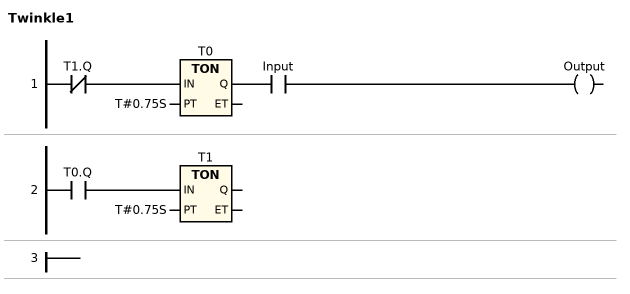
[picture p120: Twinkle1 (LD)]
_LD_ (* Ladder Diagram *)
NETWORK 1
	[/T1.Q] - T0:TON(IN: *, PT: T#0.75S) - [Input] --- (Output)
NETWORK 2
	[T0.Q] - T1:TON(IN: *, PT: T#0.75S)
NETWORK 3
	*
_END_LD_
(* the same logic as Structured Text *)
(* Network 1 *)
T0(IN := NOT T1.Q, PT := T#0.75S);
Output := T0.Q AND Input;
(* Network 2 *)
T1(IN := T0.Q, PT := T#0.75S);
(* Network 3 *)
END_FUNCTION_BLOCK

(* POU Test_Part_pro/Coord_Test, ST *)
PROGRAM Coord_Test
VAR

END_VAR
DTest[0]:=A11_W2;
DTest[1]:=A11_W3;
DTest[2]:=A11_W4;
DTest[3]:=A11_W5;

DTest00[0]:=A11_W6;
DTest00[1]:=A11_W7;
DTest00[2]:=A11_W8;
DTest00[3]:=A11_W9;

DTest0[0]:=A1_W2;
DTest0[1]:=A1_W3;
DTest0[2]:=A1_W4;
DTest0[3]:=A1_W5;

DTest10[0]:=A1_W6;
DTest10[1]:=A1_W7;
DTest10[2]:=A1_W8;
DTest10[3]:=A1_W9;


(*上下气缸对调--------------------------------------------------------程序*)
IF BU2 THEN (*滑台切换1------------------按钮*)
Y1_6:=TRUE;
Y1_7:=TRUE;
BU2:=FALSE;
END_IF

IF BU1 THEN(*滑台切换1------------------按钮*)
Y1_6:=FALSE;
Y1_7:=FALSE;
BU1:=FALSE;
END_IF
END_PROGRAM

(* POU Test_Part_pro/Y09LOOP, LD *)
PROGRAM Y09LOOP
VAR
	M0: BOOL;
	TT1: TON;
	M1: BOOL;
	TT2: TON;
END_VAR
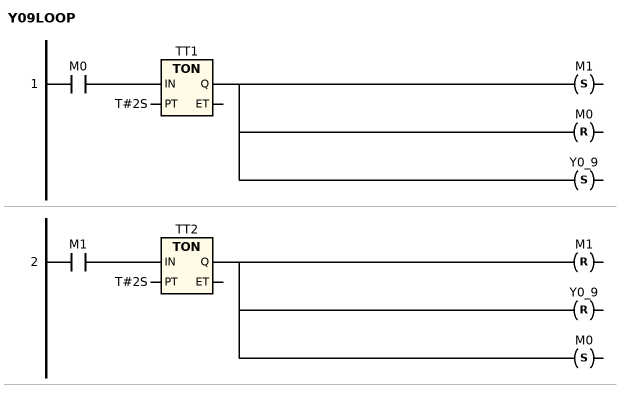
_LD_ (* Ladder Diagram *)
NETWORK 1
	[M0] - TT1:TON(IN: *, PT: T#2S) --- (S M1) (R M0) (S Y0_9)
NETWORK 2
	[M1] - TT2:TON(IN: *, PT: T#2S) --- (R M1) (R Y0_9) (S M0)
_END_LD_
(* the same logic as Structured Text *)
(* Network 1 *)
TT1(IN := M0, PT := T#2S);
IF TT1.Q THEN M1 := TRUE; M0 := FALSE; Y0_9 := TRUE; END_IF;
(* Network 2 *)
TT2(IN := M1, PT := T#2S);
IF TT2.Q THEN M1 := FALSE; Y0_9 := FALSE; M0 := TRUE; END_IF;
END_PROGRAM

(* POU Test_Part_pro/Camera_Test, ST *)
PROGRAM Camera_Test
VAR
	UP1: R_TRIG;
	UP2: R_TRIG;
	UP3: R_TRIG;
	UP4: R_TRIG;
	UP5: R_TRIG;
	UP6: R_TRIG;
	UP7: R_TRIG;
	UP8: R_TRIG;
	UP9: R_TRIG;
	number:INT;
	step:INT;
	aaaa: BOOL;

END_VAR
UP1(CLK:=Test_Camera_Run , Q=> );


CASE step OF
0:
 IF UP1.Q THEN
number:=0;
step:=10;
END_IF


10:(*跑坐标*)
UP2(CLK:=aaaa OR X4_6 , Q=> );
IF UP2.Q THEN
D1:=DTest0[number];
Axis1_MoveAbsolute:=TRUE;
END_IF
IF Axis1_Abs_Function.Done THEN
Axis1_MoveAbsolute:=FALSE;
step:=50;
END_IF

50:
UP2(CLK:=aaaa OR X4_6 , Q=> );
IF UP2.Q THEN
D1:=DTest10[number];
Axis1_MoveAbsolute:=TRUE;
END_IF
IF Axis1_Abs_Function.Done THEN
Axis1_MoveAbsolute:=FALSE;
number:=number+1;
step:=10;
END_IF
END_CASE


IF number=4 THEN
number:=0;
END_IF


IF Test_Camera_Run1 OR  Total_Emergency  THEN
Test_Camera_Run:=FALSE;
step:=0;
number:=0;
END_IF
END_PROGRAM

(* POU Test_Part_pro/Camera_Test_1, ST *)
PROGRAM Camera_Test_1
VAR
	UP1: R_TRIG;
	UP2: R_TRIG;
	UP3: R_TRIG;
	UP4: R_TRIG;
	UP5: R_TRIG;
	UP6: R_TRIG;
	UP7: R_TRIG;
	UP8: R_TRIG;
	UP9: R_TRIG;
	number:INT;
	step:INT;

	aaaa: BOOL;
	ss:INT;


END_VAR
UP1(CLK:=Test_Camera_Run1 , Q=> );


CASE step OF
0:
 IF UP1.Q THEN
number:=0;
step:=10;
END_IF


10:(*跑坐标*)
UP2(CLK:=aaaa OR X4_6 , Q=> );
IF UP2.Q THEN
D1_1:=DTest[number];
Axis11_MoveAbsolute:=TRUE;
END_IF
IF Axis11_Abs_Function.Done THEN
Axis11_MoveAbsolute:=FALSE;
step:=50;
END_IF

50:
UP2(CLK:=aaaa OR X4_6 , Q=> );
IF UP2.Q THEN
D1_1:=DTest00[number];
Axis11_MoveAbsolute:=TRUE;
END_IF
IF Axis11_Abs_Function.Done THEN
Axis11_MoveAbsolute:=FALSE;
number:=number+1;
step:=10;
END_IF
END_CASE


IF number=4 THEN
number:=0;
END_IF


IF Test_Camera_Run OR  Total_Emergency  THEN
Test_Camera_Run1:=FALSE;
step:=0;
number:=0;
END_IF
END_PROGRAM

(* POU Test_Part_pro/Camera_Test_loop, ST *)
PROGRAM Camera_Test_loop
VAR
	UP1: R_TRIG;
	UP2: R_TRIG;
	UP3: R_TRIG;
	UP4: R_TRIG;
	UP5: R_TRIG;
	UP6: R_TRIG;
	UP7: R_TRIG;
	UP8: R_TRIG;
	UP9: R_TRIG;
	number:INT;
	step:INT;
	aaaa: BOOL;


END_VAR
(*滑台1特殊操作程序*)


UP1(CLK:=Test_Camera_Run_loop , Q=> );


CASE step OF
0:
 IF UP1.Q THEN
number:=0;
step:=10;
END_IF


10:(*跑坐标*)
UP2(CLK:=aaaa OR X4_6 OR All_Rset  , Q=> );
IF UP2.Q THEN
D1:=DTest0[number];
Axis1_MoveAbsolute:=TRUE;
END_IF
IF Axis1_Abs_Function.Done THEN
Axis1_MoveAbsolute:=FALSE;
number:=number+1;
step:=20;
END_IF

20:
IF number<4 THEN
step:=10;
END_IF
IF number=4 THEN
number:=0;
step:=30;
END_IF

30:
UP2(CLK:=aaaa OR X4_6 OR All_Rset , Q=> );
IF UP2.Q THEN
D1:=DTest10[number];
Axis1_MoveAbsolute:=TRUE;
END_IF
IF Axis1_Abs_Function.Done THEN
Axis1_MoveAbsolute:=FALSE;
number:=number+1;
step:=40;
END_IF

40:
IF number<4 THEN
step:=30;
END_IF
IF number=4 THEN
number:=0;
step:=10;
END_IF

(*
50:
UP2(CLK:=aaaa OR X4_6 OR All_Rset , Q=> );
IF UP2.Q THEN
D1:=Debug1[number];
Axis1_MoveAbsolute:=TRUE;
END_IF
IF Axis1_Abs_Function.Done THEN
Axis1_MoveAbsolute:=FALSE;
number:=number+1;
step:=60;
END_IF

60:
IF number<4 THEN
step:=50;
END_IF
IF number=4 THEN
number:=0;
step:=10;
END_IF*)

END_CASE

IF   Total_Emergency OR Rset_Test1  THEN
Test_Camera_Run_loop:=FALSE;
step:=0;
number:=0;
END_IF
END_PROGRAM

(* POU Test_Part_pro/Camera_Test_loop_1, ST *)
PROGRAM Camera_Test_loop_1
VAR
	UP1: R_TRIG;
	UP2: R_TRIG;
	UP3: R_TRIG;
	UP4: R_TRIG;
	UP5: R_TRIG;
	UP6: R_TRIG;
	UP7: R_TRIG;
	UP8: R_TRIG;
	UP9: R_TRIG;
	number:INT;
	step:INT;
	aaaa: BOOL;



END_VAR
(*滑台2特殊操作程序*)


UP1(CLK:=Test_Camera_Run_loop1 , Q=> );


CASE step OF
0:
 IF UP1.Q   THEN
number:=0;
step:=10;
END_IF


10:(*跑坐标*)
UP2(CLK:=aaaa OR X4_6 OR All_Rset , Q=> );
IF UP2.Q THEN
D1_1:=DTest[number];
Axis11_MoveAbsolute:=TRUE;
END_IF
IF Axis11_Abs_Function.Done THEN
Axis11_MoveAbsolute:=FALSE;
number:=number+1;
step:=20;
END_IF

20:
IF number<4 THEN
step:=10;
END_IF
IF number=4 THEN
number:=0;
step:=30;
END_IF

30:
UP2(CLK:=aaaa OR X4_6 OR All_Rset , Q=> );
IF UP2.Q THEN
D1_1:=DTest00[number];
Axis11_MoveAbsolute:=TRUE;
END_IF
IF Axis11_Abs_Function.Done THEN
Axis11_MoveAbsolute:=FALSE;
number:=number+1;
step:=40;
END_IF

40:
IF number<4 THEN
step:=30;
END_IF
IF number=4 THEN
number:=0;
step:=10;
END_IF

END_CASE

IF   Total_Emergency OR Rset_Test2  THEN
Test_Camera_Run_loop1:=FALSE;
step:=0;
number:=0;
END_IF
END_PROGRAM

(* POU Test_Part_pro/Rolling_Part_1, ST *)
PROGRAM Rolling_Part_1
VAR
	step: INT;
	bak_step:INT;
	rt_hold: R_TRIG;
	UP1: R_TRIG;
	T1: TON;
	T2:TON;

	T6: TON;

END_VAR
UP1(CLK:= Rolling_Part_Run_Test   , Q=> );

CASE step OF
0:
 IF UP1.Q  THEN
step:=10;
END_IF

10:(*滚压部分开始动作*)
(*判断机械手是否放好料---------放好之后，进行滚压动作，询问右移载是否可以送料，可送料之后，给出料，同时，发出，给料完成信号*)
IF  Rolling_Once_Run THEN
	step:=20;
END_IF

20:(*无料的操作*)
D10:=A10_W2;
Axis10_MoveAbsolute:=TRUE;
IF Axis10_Abs_Function.Done THEN
Axis10_MoveAbsolute:=FALSE;
step:=31;
END_IF


31:
	IF Empty_Pro THEN

	step:=30;
	ELSE
Y0_12:=TRUE;(*滚压平台*)
	step:=30;
END_IF


30:(*等待机械手2.放料*)
IF Robot2_Push_Finish OR Rolling_Once_Run THEN
Rolling_Number:=0;
Y0_10:=TRUE;(*推入气缸*)
step:=50;
END_IF


50:
IF X2_16 THEN
Y0_9:=TRUE;
Y0_11:=TRUE;
step:=60;
END_IF

60:
IF X3_2  THEN(*压合气缸到位，等待滚压*)
step:=70;
END_IF

70:
D10_1:=A10_W1;(*出去位置*)(*滚压低速*)
Axis10_MoveAbsolute1:=TRUE;
IF Axis10_Abs_Function1.Done THEN
Axis10_MoveAbsolute1:=FALSE;
Y0_9:=FALSE;
Y0_11:=FALSE;
step:=78;
END_IF

78:
IF X3_3 THEN
step:=80;
END_IF

80:
D10:=A10_W2;
Axis10_MoveAbsolute:=TRUE;
IF Axis10_Abs_Function.Done THEN
Axis10_MoveAbsolute:=FALSE;
Rolling_Number:=Rolling_Number+1;
step:=90;
END_IF

90:
IF Rolling_Number>=Set_Rolling_Number THEN
Rolling_Number:=0;

Y0_9:=FALSE;
step:=100;(*次数满足，跳转*)
ELSE
step:=50;
END_IF

100:
IF X3_3 THEN
Y0_10:=FALSE;
step:=110;
END_IF

110:
IF X3_1 THEN
step:=120;
END_IF

120:(*滚压回到安全位置------询问是否可以扣料*)
IF Process_4_Can_Push OR Rolling_Pushor_NOT THEN

Y0_13:=TRUE;(*翻转动作开始动作*)
step:=130;
ELSE
Rolling_Once_Run:=FALSE;
step:=10;
END_IF


130:
IF X3_4 THEN

step:=131;
END_IF

131:
IF Empty_Pro THEN
step:=139;
ELSE
Y0_14:=TRUE;(*右真空吸开始吸取*)
y0_1:=TRUE;
step:=139;
END_IF


139:
T6(IN:=TRUE , PT:=t#0.15s , Q=> , ET=> );
   IF T6.Q   THEN
T6(IN:=FALSE, PT:=t#0.15S , Q=> , ET=> );
Y0_12:=FALSE;
step:=140;
END_IF

140:
T2(IN:=TRUE , PT:=t#0.1s , Q=> , ET=> );
   IF T2.Q   THEN
T2(IN:=FALSE, PT:=t#0.1S , Q=> , ET=> );
Y0_13:=FALSE;
step:=150;
END_IF

150:
IF X3_5 THEN(*翻转结构�--------完成------告知机械手*)
Rolling_Once_Run:=FALSE;
step:=10;
END_IF


END_CASE





IF Total_Emergency  OR Rolling_Part_Run_Test_OFF  THEN
Rolling_Part_Run:=FALSE;
Process_3_Set_Finish:=FALSE;
Process_3_Can_Push:=FALSE;

rolling_have_liao:=FALSE;
Process_3_Can_Push:=FALSE;
Wait_Robot_Push:=FALSE;
Robot2_Push_Finish:=FALSE;
Rolling_Number:=0;
Process_4_Can_Push:=FALSE;
Process_3_Set_Finish:=FALSE;
Rolling_Part_Run_Test:=FALSE;

bak_step:=0;
step:=0;
END_IF
END_PROGRAM

(* POU Run_Main_Folder/Barcode/Brd_Run, ST *)
PROGRAM Brd_Run
VAR
	UP1: R_TRIG;
	step: INT;
	bak_step:INT;
	rt_hold: R_TRIG;

	T1:TON;
	T2:TON;
	T3:TON;
	T4:TON;
	T5:TON;
	T6:TON;
	loopTimes:INT;
END_VAR

VAR_INPUT
	bstart1: BOOL;
	bhold1: BOOL;
	breset1: BOOL;

END_VAR
(*条码部分程序*)

(*等待启动*)
UP1(CLK:=Brd_Start_Run , Q=> );

CASE step OF

0:
 IF UP1.Q THEN
	Y101_5:=TRUE;
	step:=10;
END_IF

10:(*等待条码到位*)
IF X101_10 THEN
	Y101_5:=FALSE;
	step:=20;
END_IF

(*取条码动作*)
20:(*至取码位*)
V24:=A24PPick;(*Z轴取料位置等待*)
V25:=A25PPick;(*U轴取料位置等待*)
V22:=A22PPick;(*Y轴取料位置等待*)
Axis24_MoveAbsolute:=TRUE;
Axis25_MoveAbsolute:=TRUE;
Axis22_MoveAbsolute:=TRUE;
IF Axis24_Abs_Function.Done AND  Axis25_Abs_Function.Done AND  Axis22_Abs_Function.Done THEN
Axis24_MoveAbsolute:=FALSE;
Axis25_MoveAbsolute:=FALSE;
Axis22_MoveAbsolute:=FALSE;
step:=30;
END_IF

30:(*取码气缸动作*)
IF NOT X101_1 THEN Y100_3:=TRUE;END_IF
IF NOT X101_2 THEN Y100_4:=TRUE;END_IF
IF NOT X101_3 THEN Y100_5:=TRUE;END_IF
IF NOT X101_4 THEN Y100_6:=TRUE;END_IF
T1(IN:=TRUE , PT:= t#0.6s );
IF T1.ET>=t#0.3s THEN(*真空吸*)
	IF NOT X101_1 THEN Y100_13:=TRUE; END_IF
	IF NOT X101_2 THEN Y100_14:=TRUE; END_IF
	IF NOT X101_3 THEN Y100_15:=TRUE; END_IF
	IF NOT X101_4 THEN Y100_16:=TRUE; END_IF
END_IF

IF T1.Q THEN
	T1(IN:=FALSE);
	step:=40;
END_IF

40:(*复位气缸*)
Y100_3:=FALSE;
Y100_4:=FALSE;
Y100_5:=FALSE;
Y100_6:=FALSE;
T2(IN:=TRUE , PT:= t#0.5s );

IF T2.Q THEN
	T2(IN:=FALSE);
	step:=50;
END_IF

50:(*判断吸取状态*)
IF X101_1 AND X101_2 AND X101_3 AND X101_4 THEN
	step:=70;
	loopTimes:=0;
ELSE
	loopTimes:=loopTimes+1;
	IF loopTimes>3 THEN
		step:=60;
	ELSE
		step:=30;
	END_IF
END_IF

60:(*多次吸取失败报警*)
loopTimes:=0;
Alarm_Pick_Barcode_Fail:=TRUE;
step:=61;

61:
T4(IN:=TRUE , PT:= t#0.5s );
IF T4.Q THEN
	T4(IN:=FALSE);
	Alarm_Pick_Barcode_Fail:=FALSE;
	Y101_5:=TRUE;
	step:=10;
END_IF

70:(*至拍摄位等待拍摄*)
V24:=A24PCam;(*Z轴拍摄位置等待*)
V25:=A25PCam;(*U轴拍摄位置等待*)
V22:=A22PCam;(*Y轴拍摄位置等待*)
Axis24_MoveAbsolute:=TRUE;
Axis25_MoveAbsolute:=TRUE;
Axis22_MoveAbsolute:=TRUE;
IF Axis24_Abs_Function.Done AND  Axis25_Abs_Function.Done AND  Axis22_Abs_Function.Done THEN
	Axis24_MoveAbsolute:=FALSE;
	Axis25_MoveAbsolute:=FALSE;
	Axis22_MoveAbsolute:=FALSE;
	Flag_Barcode_Need_Cam:=TRUE;
	step:=80;
END_IF

80:(*接受可以贴合指令*)
IF Flag_Barcode_Can_Fit=TRUE THEN
	Flag_Barcode_Can_Fit:=FALSE;
	step:=90;
END_IF

90:(*开始贴合*)
V24:=A24PDrop;(*Z轴贴合位置等待*)
V25:=A25PDrop;(*U轴贴合位置等待*)
V22:=A22PDrop;(*Y轴贴合位置等待*)
Axis24_MoveAbsolute:=TRUE;
Axis25_MoveAbsolute:=TRUE;
Axis22_MoveAbsolute:=TRUE;
IF Axis24_Abs_Function.Done AND  Axis25_Abs_Function.Done AND  Axis22_Abs_Function.Done THEN
	Axis24_MoveAbsolute:=FALSE;
	Axis25_MoveAbsolute:=FALSE;
	Axis22_MoveAbsolute:=FALSE;
	step:=100;
END_IF

100:(*张开气缸*)
Y101_6:=TRUE;
T5(IN:=TRUE , PT:= t#0.5s );
IF T5.Q THEN
	T5(IN:=FALSE);
	step:=110;
END_IF

110:
Y100_3:=TRUE;
Y100_4:=TRUE;
Y100_5:=TRUE;
Y100_6:=TRUE;
T6(IN:=TRUE , PT:= t#0.6s );
IF T6.ET>=t#0.4s THEN
	Y100_13:=FALSE;
	Y100_14:=FALSE;
	Y100_15:=FALSE;
	Y100_16:=FALSE;
	Y101_1:=TRUE;
	Y101_2:=TRUE;
	Y101_3:=TRUE;
	Y101_4:=TRUE;
END_IF

IF T6.Q THEN
	T6(IN:=FALSE);
	Y101_1:=FALSE;
	Y101_2:=FALSE;
	Y101_3:=FALSE;
	Y101_4:=FALSE;
	Y100_3:=FALSE;
	Y100_4:=FALSE;
	Y100_5:=FALSE;
	Y100_6:=FALSE;
	step:=120;
END_IF

120:
V24:=A24PSafe;(*Z轴贴合位置等待*)
V25:=A25PPick;(*U轴贴合位置等待*)
V22:=A22PPick;(*Y轴贴合位置等待*)
Axis24_MoveAbsolute:=TRUE;
Axis25_MoveAbsolute:=TRUE;
Axis22_MoveAbsolute:=TRUE;
IF Axis24_Abs_Function.Done AND  Axis25_Abs_Function.Done AND  Axis22_Abs_Function.Done THEN
	Axis24_MoveAbsolute:=FALSE;
	Axis25_MoveAbsolute:=FALSE;
	Axis22_MoveAbsolute:=FALSE;
	Flag_Barcode_Fit_Finish:=TRUE;
	step:=10;
END_IF

300:
IF bstart1   AND NOT Total_Axis_Error AND NOT total_pausestatus  THEN
	step:=bak_step;
END_IF;

END_CASE

rt_hold(CLK:=( Total_Axis_Error OR  bhold1) , Q=> ); (*暂停状态*)
IF step<>0 AND step<>300   AND  rt_hold.Q THEN
     bak_step:=step;
     step:=300;
END_IF

IF Total_Emergency THEN
	loopTimes:=0;
	Flag_Barcode_Can_Fit:=FALSE;
	Flag_Barcode_Fit_Finish:=FALSE;
	Flag_Barcode_Need_Cam:=FALSE;
	Y101_5:=FALSE;
	Y101_6:=FALSE;
	Y100_3:=FALSE;
	Y100_4:=FALSE;
	Y100_5:=FALSE;
	Y100_6:=FALSE;
	Y100_13:=FALSE;
	Y100_14:=FALSE;
	Y100_15:=FALSE;
	Y100_16:=FALSE;
	Y101_1:=FALSE;
	Y101_2:=FALSE;
	Y101_3:=FALSE;
	Y101_4:=FALSE;
	bak_step:=0;
	step:=0;
END_IF
END_PROGRAM

(* POU Other_Folder/Akam_Stop_Message/Initialization_Folder/New_IniRun, ST *)
PROGRAM New_IniRun
VAR
	step: INT;
	bak_step:INT;
	rt_hold: R_TRIG;
	M1: BOOL;

	T1: TON;
	T2:TON;



END_VAR

VAR_INPUT
	bstart1: BOOL;
	bhold1: BOOL;
	breset1: BOOL;

END_VAR
(*数据保存*)
IF Save_Button THEN
Save_Par(NETID:='',port:=801,start:=TRUE,tmout:=T#1s);
END_IF
IF NOT Save_Par.BUSY  THEN
Save_Button:=FALSE;
Save_Par(NETID:='',port:=801,start:=FALSE,tmout:=T#1s);
END_IF

(*当出现回原点没有时，需要初始化*)
IF NOT Axis1_BackHome_OK OR NOT  Axis2_BackHome_OK OR NOT Axis3_BackHome_OK OR NOT Axis4_BackHome_OK OR NOT Axis5_BackHome_OK
	OR NOT Axis6_BackHome_OK OR NOT Axis7_BackHome_OK OR NOT Axis8_BackHome_OK OR NOT Axis9_BackHome_OK OR NOT Axis10_BackHome_OK OR NOT Axis11_BackHome_OK
	OR NOT Axis21_Backhome_Ok OR NOT Axis22_Backhome_Ok OR NOT Axis23_Backhome_Ok OR NOT Axis24_Backhome_Ok OR NOT Axis25_Backhome_Ok

	 THEN
;(*判断是否需要回原点----------------------------------------------------*)
END_IF
(*---------------------------------------------------------------------------初始化开始流程---------------------------------------------------------------------------------*)
CASE step OF
0:
Need_Ini:=TRUE;(*此时寻妖初始化*)
(*进入初始化流程*)
step:=10;

10:(*判断是否需要初始化*)
IF Need_Ini AND NOT Total_Axis_Error AND NOT Debug_Model   THEN (*当需要初始化的时候，复位所有原点ok信号*)
	Axis1_BackHome_OK:=FALSE;
Axis2_BackHome_OK:=FALSE;
Axis3_BackHome_OK:=FALSE;
Axis4_BackHome_OK:=FALSE;
Axis5_BackHome_OK:=FALSE;
Axis6_BackHome_OK:=FALSE;
Axis7_BackHome_OK:=FALSE;
Axis8_BackHome_OK:=FALSE;
Axis9_BackHome_OK:=FALSE;
Axis10_BackHome_OK:=FALSE;
Axis11_BackHome_OK:=FALSE;

Axis21_BackHome_OK:=FALSE;
Axis22_BackHome_OK:=FALSE;
Axis23_BackHome_OK:=FALSE;
Axis24_BackHome_OK:=FALSE;
Axis25_BackHome_OK:=FALSE;

step:=20;
END_IF

20:(*等待复位按钮操作，复位报警等状态*)
IF (X4_6 OR All_Rset ) AND Need_Ini AND X100_14 THEN
	IF Total_Axis_Error THEN
	M1:=TRUE;(*no use*)(*上位机提示电机报警问题，需要初始化*)
	END_IF
	IF NOT Total_Axis_Error THEN
	step:=30;
	END_IF
END_IF;

30:(*启动按下的处理开始进入初始化过中。。。。。。*)
IF (X4_4 OR All_Start) AND NOT Total_Axis_Error AND NOT Debug_Model THEN
Need_Ini:=FALSE;
IsIniing:=TRUE;(*初始化中ing*)
M101:=TRUE;(*初始化中，速度为中速*)
Axis1_Poweron:=TRUE;
Axis2_Poweron:=TRUE;
Axis3_Poweron:=TRUE;
Axis4_Poweron:=TRUE;
Axis5_Poweron:=TRUE;
Axis6_Poweron:=TRUE;
Axis7_Poweron:=TRUE;
Axis8_Poweron:=TRUE;
Axis9_Poweron:=TRUE;
Axis10_Poweron:=TRUE;
Axis11_Poweron:=TRUE;

Axis21_Poweron:=TRUE;
Axis22_Poweron:=TRUE;
Axis23_Poweron:=TRUE;
Axis24_Poweron:=TRUE;
Axis25_Poweron:=TRUE;

step:=39;
END_IF

39:
(*滑台气缸上下，如果在同一高度，则说明不存在重叠部分，可复位气缸*)
IF (X4_11 AND X4_13) OR (X4_12 AND X4_14)  AND X2_6 THEN
Y1_6:=FALSE;
Y1_7:=FALSE;
step:=40;
ELSE
step:=40;
END_IF


40:(*气缸复位状态保留*)


Y0_12:=FALSE;



(******************** AND  *****************************)

Y0_7:=FALSE;(*左上下气缸*)
Y0_2:=FALSE;Y0_5:=FALSE;
Y0_9:=FALSE;(*滚压气缸复位*)
Y1_1:=FALSE;(*右上下气缸*)
Y1_3:=FALSE;
IF X2_13  AND X3_11 THEN
	step:=50;(*初步气缸复位*)
END_IF

50:
Y0_6:=FALSE;(*左平移气缸复位*)
Y0_11:=FALSE;(*滚压部分下压气缸复位*)
Y0_16:=FALSE;(*右平移气缸复位*)
T1(IN:=TRUE , PT:=t#1s , Q=> , ET=> );
IF T1.Q AND X2_11 AND X3_9 THEN
T1(IN:=FALSE , PT:=t#1s , Q=> , ET=> );
step:=60;(*无感气缸*)
END_IF

60:(*复位滚压气缸部分气缸，推入气缸，和翻转气缸*)
Y0_10:=FALSE;
IF X3_1 THEN
step:=70;
END_IF

70:(*翻转气缸复位*)
Y0_13:=FALSE;
IF X3_5 THEN
step:=80;
END_IF

80:(*上电延时*)
T2(IN:=TRUE , PT:=t#1s , Q=> , ET=> );
IF T2.Q  AND NOT Total_Pause THEN
T2(IN:=FALSE , PT:=t#1s , Q=> , ET=> );
step:=90;
END_IF

90:
home_backing:=TRUE;
IF NOT Axis3_BackHome_OK OR NOT Axis6_BackHome_OK OR NOT Axis7_BackHome_OK OR NOT Axis8_BackHome_OK OR NOT Axis9_BackHome_OK THEN
step:=100;
ELSE
step:=110;(*当喂料都已经回过原点，则不需要回原点*)
END_IF


100:(*判断是否都需要回原点*)(*喂料部分回原点*)
Axis3_BackHome_trigger:=TRUE;(**)
Axis6_BackHome_trigger:=TRUE;(**)
Axis7_BackHome_trigger:=TRUE;(**)
Axis8_BackHome_trigger:=TRUE;(**)
Axis9_BackHome_trigger:=TRUE;
IF Axis3_BackHome_OK AND Axis6_BackHome_OK AND Axis7_BackHome_OK AND Axis8_BackHome_OK AND Axis9_BackHome_OK  THEN
Axis3_BackHome_trigger:=FALSE;(**)
Axis6_BackHome_trigger:=FALSE;(**)
Axis7_BackHome_trigger:=FALSE;(**)
Axis8_BackHome_trigger:=FALSE;(**)
Axis9_BackHome_trigger:=FALSE;
step:=101;
END_IF

101:(*升降回到初始位置*)
D3:=D300;(*进料初始位置，在下面*)
D6:=D600;(*上升初始位置，在下面*)
D7:=D700;(*下降初始位置，在下面*)
D8:=D800;(*上升初始位置，在下面*)
D9:=D900;(*下降初始位置，在下面*)
Axis3_MoveAbsolute:=TRUE;
Axis6_MoveAbsolute:=TRUE;
Axis7_MoveAbsolute:=TRUE;
Axis8_MoveAbsolute:=TRUE;
Axis9_MoveAbsolute:=TRUE;
IF Axis3_Abs_Function.Done AND Axis6_Abs_Function.Done AND Axis7_Abs_Function.Done AND Axis8_Abs_Function.Done AND Axis9_Abs_Function.Done  THEN
Axis3_MoveAbsolute:=FALSE;
Axis6_MoveAbsolute:=FALSE;
Axis7_MoveAbsolute:=FALSE;
Axis8_MoveAbsolute:=FALSE;
Axis9_MoveAbsolute:=FALSE;
step:=102;  (*初始都在下面*)
END_IF

102:(*Z轴撕膜电机回原*)
Axis5_BackHome_trigger:=TRUE;
IF Axis5_BackHome_OK THEN
Axis5_BackHome_trigger:=FALSE;
step:=103;
END_IF

103:
D5:=A5_W0;(*Z轴回到初始位置*)
Axis5_MoveAbsolute:=TRUE;
IF Axis5_Abs_Function.Done THEN
Y0_4:=FALSE;
Y1_4:=FALSE;
Axis5_MoveAbsolute:=FALSE;
step:=105;
END_IF

(*滚压和条码z回原点*)
105:
Axis23_BackHome_trigger:=TRUE;
Axis24_BackHome_trigger:=TRUE;
IF Axis23_BackHome_OK  AND Axis24_BackHome_OK  THEN
	Axis23_BackHome_trigger:=FALSE;
	Axis24_BackHome_trigger:=FALSE;
	step:=106;
END_IF


106:
Axis25_BackHome_trigger:=TRUE;
IF Axis25_BackHome_OK THEN
	Axis25_BackHome_trigger:=FALSE;
	step:=110;
END_IF

110:(*其余轴回原点*)
Axis1_BackHome_trigger:=TRUE;
Axis11_BackHome_trigger:=TRUE;
Axis2_BackHome_trigger:=TRUE;
Axis4_BackHome_trigger:=TRUE;
Axis10_BackHome_trigger:=TRUE;

Axis21_BackHome_trigger:=TRUE;
Axis22_BackHome_trigger:=TRUE;
IF Axis1_BackHome_OK AND Axis2_BackHome_OK AND Axis4_BackHome_OK  AND Axis10_BackHome_OK AND Axis11_BackHome_OK   AND Axis21_BackHome_OK   AND Axis22_BackHome_OK  THEN
Axis1_BackHome_trigger:=FALSE;
Axis2_BackHome_trigger:=FALSE;
Axis4_BackHome_trigger:=FALSE;
Axis10_BackHome_trigger:=FALSE;
Axis11_BackHome_trigger:=FALSE;
Axis21_BackHome_trigger:=FALSE;
Axis22_BackHome_trigger:=FALSE;
step:=120;
END_IF

120:(*移载等轴的回到初始位置*)
D1:=A1_W0;
D1_1:=A11_W0+300;(*为了保证回原点之后，滑台1气缸在下面，滑台2气缸在上面，则需要，错开初始位置*)
D2:=A2_W0;
D4:=A4_W0;
D10:=A10_W0;
Axis1_MoveAbsolute:=TRUE;
Axis2_MoveAbsolute:=TRUE;
Axis4_MoveAbsolute:=TRUE;
Axis10_MoveAbsolute:=TRUE;
Axis11_MoveAbsolute:=TRUE;
IF Axis1_Abs_Function.Done AND Axis2_Abs_Function.Done AND Axis4_Abs_Function.Done  AND Axis10_Abs_Function.Done AND Axis11_Abs_Function.Done  THEN
Axis1_MoveAbsolute:=FALSE;
Axis2_MoveAbsolute:=FALSE;
Axis4_MoveAbsolute:=FALSE;
Axis10_MoveAbsolute:=FALSE;
Axis11_MoveAbsolute:=FALSE;
home_backing:=FALSE;
Y1_6:=FALSE;(*最终保证，滑台1在上面，滑台2气缸在下面*)
Y1_7:=FALSE;
step:=121;
END_IF


121:
IF  X4_11 THEN(*最终结果，传感器检测*)
step:=122;
END_IF

122:
D1_1:=A11_W0;
Axis11_MoveAbsolute:=TRUE;
IF  Axis11_Abs_Function.Done THEN
Axis11_MoveAbsolute:=FALSE;
step:=130;
END_IF


130:(*其余需要初始化的状态*)

IsIniing:=FALSE;
Model_Choose:=TRUE;(*模式选择*)
step:=140;

140:
(*模式选选择，直接按钮，启动程序，当选上位机选择调试模式，同时按下启动按钮，则进入调试模式*)
IF NOT Debug_Model AND (X4_4 OR All_Start) THEN
	Model_Choose:=FALSE;(*模式选择*)
Product_Film_Handel_Run:=TRUE;
Left_Translation_Run_1:=TRUE;
Left_Translation_Run_2:=TRUE;
Right_Translation_Run:=TRUE;
Rolling_Part_Run:=TRUE;
Right_Carry_Run:=TRUE;
Left_Carry_Run:=TRUE;
Liftin_Feed_1_Run:=TRUE;
Liftin_Feed_Left_1_Run:=TRUE;
Liftin_Feed_Left_2_Run:=TRUE;
Liftin_Feed_Right_1_Run:=TRUE;
Liftin_Feed_Right_2_Run:=TRUE;
M101:=TRUE;
Debug_Model:=FALSE;


Positive2_Safe:=TRUE;
Positive3_Safe:=TRUE;
Positive_Wait_Safe:=TRUE;
Positive_Fit_Safe1:=TRUE;
Positive_Fit_Safe2:=TRUE;
Positive_Fit_Safe3:=TRUE;
Positive_Fit_Safe4:=TRUE;
Positive_Camera_Safe1:=TRUE;
Positive_Camera_Safe2:=TRUE;
Positive_Camera_Safe3:=TRUE;
Positive_Camera_Safe4:=TRUE;



runing:=TRUE;
	step:=150;
END_IF
IF Debug_Model AND (X4_4 OR All_Start) THEN
	M100:=TRUE;(*调试模式下低速*)
	Model_Choose:=FALSE;(*模式选择*)
	Axis1_debug_trigger:=TRUE;
Axis1_debug_trigger:=TRUE;
Axis2_debug_trigger:=TRUE;
Axis3_debug_trigger:=TRUE;
Axis4_debug_trigger:=TRUE;
Axis5_debug_trigger:=TRUE;
Axis6_debug_trigger:=TRUE;
Axis7_debug_trigger:=TRUE;
Axis8_debug_trigger:=TRUE;
Axis9_debug_trigger:=TRUE;
Axis10_debug_trigger:=TRUE;
Axis11_debug_trigger:=TRUE;
(*其余调试模式*)
 step:=160;
END_IF

150:(*运行模式下的死循环*)
;


160:
(*调试模式下的死循环，等待调试模式借宿，重新开始初始化*)
IF NOT Debug_Model THEN
Need_Ini:=TRUE;
 	    bak_step:=0;
	step:=0;
END_IF



300:(*外部输入启动*)
    IF bstart1   AND NOT Total_Axis_Error AND NOT total_pausestatus THEN
	step:=bak_step;
END_IF;
END_CASE;



(*触发暂停的外部输入*)
rt_hold(CLK:=( Total_Axis_Error OR  bhold1) , Q=> ); (*暂停状态*)
IF step<>0 AND step<>300   AND  rt_hold.Q THEN
     bak_step:=step;
     step:=300;
END_IF

(*急停处理*)
IF Total_Emergency THEN
debug_FLIG:=FALSE;
M100:=FALSE;
M101:=FALSE;
M102:=FALSE;
IsIniing:=FALSE;
runing:=FALSE;
home_backing:=FALSE;
Model_Choose:=FALSE;(*模式选择*)


Debug_Model:=FALSE;
Positive2_Safe:=FALSE;
Positive3_Safe:=FALSE;
Positive_Wait_Safe:=FALSE;


bak_step:=0;
step:=0;
END_IF


(*与debug1中的梯形图一起使用，当不在应该调试模式下的时候，按下调试按钮，自动复位--------详见------debug1----------*)
IF step<>160 AND step<>140 AND step<>300  THEN
debug_FLIG:=FALSE;
ELSE
debug_FLIG:=TRUE;
END_IF
END_PROGRAM

(* POU Run_Main_Folder/Film_Handel/Film_Handel_Pro_1, ST *)
PROGRAM Film_Handel_Pro_1
VAR
	DrawFailTimes:INT;
	UP1: R_TRIG;
	step: INT;
	bak_step:INT;
	rt_hold: R_TRIG;
	T1: TON;
	T2: TON;
	T3: TON;
	T4: TON;

	T5: TON;
	T6: TON;


	T9: TON;
	T10: TON;
	T100: TON;
	T101: TON;
	T102:TON;

	T103: TON;
	T104: TON;
	T99: TON;
END_VAR

VAR_INPUT
	bstart1: BOOL;
	bhold1: BOOL;
	breset1: BOOL;

END_VAR
(*撕膜部分程序*)

UP1(CLK:=Product_Film_Handel_Run , Q=> );

(*X_Z轴撕膜动作----------------------------------------
等待上料完成-------------------取料，到工作平台
等待平台到位信号--------------------取料过程中夹膜，放入平台
等待形成真空--------------------撕膜动作一体---------------
撕膜完成信号给出---------------------------------丢膜--------
丢膜完成---------------------再去取料工位，等待上料完成信号*)


CASE step OF
0:
 IF UP1.Q THEN
step:=10;
END_IF

10:(*撕膜部分开始动作*)
D4:=A4_W1;(*取料位置等待*)
Axis4_MoveAbsolute:=TRUE;
IF Axis4_Abs_Function.Done THEN
Axis4_MoveAbsolute:=FALSE;
Y100_1:=FALSE;
step:=9;
END_IF

9:
T6(IN:=TRUE , PT:=t#2s , Q=> , ET=> );
IF T1.Q AND NOT Total_Pause  THEN
	T6(IN:=FALSE, PT:=t#2S , Q=> , ET=> );
	step:=11;
END_IF

11:
IF X100_6 THEN
V21:=A21PPick1;
ELSE
V21:=A21PPick2;
END_IF
step:=12;

12:
Axis21_MoveAbsolute:=TRUE;
IF Axis21_Abs_Function.Done THEN
Axis21_MoveAbsolute:=FALSE;
step:=20;
END_IF


20: (*判断喂料1是否完成*)
IF Feed_1_Finish THEN
Feed_1_Finish:=FALSE;
step:=30;
END_IF
IF X100_6 AND V21=A21PPick2
THEN step:=11;
END_IF
IF X100_7 AND V21=A21PPick1
THEN step:=11;
END_IF


30:(*K可取料*)
D5:=A5_W1;
Axis5_MoveAbsolute:=TRUE;
IF Axis5_Abs_Function.Done THEN
Axis5_MoveAbsolute:=FALSE;
step:=40;
Y0_3:=TRUE;
END_IF

40:(*到达取料工位，准备真空吸*)
T1(IN:=TRUE , PT:=t#0.4s , Q=> , ET=> );
   IF T1.Q AND NOT Total_Pause  THEN
T1(IN:=FALSE, PT:=t#0.4S , Q=> , ET=> );
step:=50;
END_IF

50:
D15_1:=100;
D5:=A5_W0;(*回到安全位置----准备去放料平台*)
Axis5_1_MoveAbsolute:=TRUE;
IF Axis5_1_Abs_Function.Done THEN
Axis5_1_MoveAbsolute:=FALSE;
step:=99;
END_IF

99:
D15_1:=450;
D5:=A5_W0+10;(*回到安全位置----准备去放料平台*)
Axis5_1_MoveAbsolute:=TRUE;
IF Axis5_1_Abs_Function.Done THEN
Axis5_1_MoveAbsolute:=FALSE;
step:=98;
END_IF

98:
D5:=A5_W0;(*回到安全位置----准备去放料平台*)
Axis5_MoveAbsolute:=TRUE;
IF Axis5_Abs_Function.Done THEN
Axis5_MoveAbsolute:=FALSE;
step:=51;
END_IF

51:
T100(IN:=TRUE , PT:=t#0.1s , Q=> , ET=> );
   IF T100.Q AND NOT Total_Pause  THEN
T100(IN:=FALSE, PT:=t#0.1S , Q=> , ET=> );
step:=52;
END_IF


52:
IF X2_7 THEN
(*取料成功告知上料喂料流程*)
DrawFailTimes:=0;
Process_1_Get_Finish:=TRUE;
Y0_4:=TRUE;
step:=60;
END_IF
IF NOT X2_7 THEN
DrawFailTimes:=1+DrawFailTimes;
	IF DrawFailTimes >=3 THEN
		Feed_1_Finish:=FALSE;
		DrawFailTimes:=0;
		Process_1_Get_Finish:=TRUE;
		Pressure_Fail_1:=TRUE;(*吸取失败报警，暂停*)
	ELSE
		Feed_1_Finish:=TRUE;

	END_IF
	Y0_3:=FALSE;
	step:=10;

END_IF
(*
先到位置，再旋转
*)
60:(*成功吸取到料*)
T102(IN:=TRUE , PT:=t#0.5s , Q=> , ET=> );
   IF T102.Q AND NOT Total_Pause  THEN
T102(IN:=FALSE, PT:=t#0.5S , Q=> , ET=> );
Y1_4:=TRUE;
Y100_1:=TRUE;(*旋转气缸*)
step:=70;
END_IF

70:
T103(IN:=TRUE , PT:=t#0.5s , Q=> , ET=> );
   IF T103.Q AND NOT Total_Pause  THEN
T103(IN:=FALSE, PT:=t#0.5S , Q=> , ET=> );
step:=80;
END_IF

80:
D4:=A4_W4;(*到放料工位，等到是否可以放料*)
Axis4_MoveAbsolute:=TRUE;
IF Axis4_Abs_Function.Done THEN
Axis4_MoveAbsolute:=FALSE;
step:=90;
END_IF

90:(*上料是否可以判断*)
IF Process_2_Can_Push1 OR Process_2_Can_Push2  THEN
step:=100;
END_IF

100:(*上料可以之后，到放料下降工位*)
D5:=A5_W4;
Axis5_MoveAbsolute:=TRUE;
IF Axis5_Abs_Function.Done THEN
Axis5_MoveAbsolute:=FALSE;
Y0_3:=FALSE;
step:=110;
END_IF

110:
T5(IN:=TRUE , PT:=t#0.4s , Q=> , ET=> );
   IF T5.Q AND NOT Total_Pause  THEN
T5(IN:=FALSE, PT:=t#0.4S , Q=> , ET=> );
step:=111;
END_IF

111:
IF Process_2_Can_Push1 THEN
Process_2_Can_Push1:=FALSE;
Y0_5:=TRUE;
step:=112;
END_IF
IF Process_2_Can_Push2 THEN
Process_2_Can_Push2:=FALSE;
Y0_2:=TRUE;
step:=112;
END_IF

112:
T99(IN:=TRUE , PT:=t#1.3s , Q=> , ET=> );
   IF T99.Q AND NOT Total_Pause  THEN
T99(IN:=FALSE, PT:=t#1.3S , Q=> , ET=> );
Process_1_Push_Finish:=TRUE;(*等待撕膜吸嘴正式脱离之后，给出，滑台吸取的状态*)
step:=120;
END_IF

120:
IF Can_Move_Film THEN(*接收到撕膜信号之后，正式开始撕膜*)
Can_Move_Film:=FALSE;
step:=130;
END_IF

130:
D15_1:=10;
D5:=A5_W5;(*撕膜Z轴上抬一点---------*)
Axis5_1_MoveAbsolute:=TRUE;
IF Axis5_1_Abs_Function.Done THEN
Axis5_1_MoveAbsolute:=FALSE;
step:=140;
END_IF

140:(*联动*)
D14_1:=62;
D15_1:=7;
D4:=A4_W5;
D5:=A5_W6;
Axis4_1_MoveAbsolute:=TRUE;
Axis5_1_MoveAbsolute:=TRUE;
IF Axis4_1_Abs_Function.Done  AND Axis5_1_Abs_Function.Done THEN
Axis4_1_MoveAbsolute:=FALSE;
Axis5_1_MoveAbsolute:=FALSE;
step:=150;
END_IF

150:(*联动结束-------------集训动作保证进入非料盘位置*)
D15_1:=70;
D5:=A5_W8;(*Z轴上抬点位*)
Axis5_1_MoveAbsolute:=TRUE;
IF  Axis5_1_Abs_Function.Done THEN
Axis5_1_MoveAbsolute:=FALSE;
Process_1_Push_Finish_Sure:=TRUE;(*给出撕膜完成信号*)
step:=160;
END_IF

160:(*丢么位置坐标*)
D4:=A4_W3;
Axis4_MoveAbsolute:=TRUE;
IF Axis4_Abs_Function.Done THEN
Axis4_MoveAbsolute:=FALSE;
step:=170;
END_IF

170:(*丢么下降位置*)
D5:=A5_W3;
Axis5_MoveAbsolute:=TRUE;
IF   Axis5_Abs_Function.Done THEN
Axis5_MoveAbsolute:=FALSE;
Y1_4:=FALSE;(*JIAZI*)
Y0_4:=FALSE;
step:=180;
END_IF

180:
T104(IN:=TRUE , PT:=t#0.7s , Q=> , ET=> );
   IF T104.Q AND NOT Total_Pause  THEN
T104(IN:=FALSE, PT:=t#0.7S , Q=> , ET=> );
Y1_10:=TRUE;
step:=190;
END_IF

190:(*丢么位置丢弃费膜，结束，到吸取料位置*)
D5:=A5_W0;
Axis5_MoveAbsolute:=TRUE;
IF Axis5_Abs_Function.Done THEN
Axis5_MoveAbsolute:=FALSE;
Y1_10:=FALSE;
step:=10;
END_IF

300:
    IF bstart1   AND NOT Total_Axis_Error AND NOT total_pausestatus  THEN
	step:=bak_step;
END_IF;
END_CASE

rt_hold(CLK:=( Total_Axis_Error OR  bhold1) , Q=> ); (*暂停状态*)
IF step<>0 AND step<>300   AND  rt_hold.Q THEN
     bak_step:=step;
     step:=300;
END_IF

IF Total_Emergency THEN
Y1_10:=FALSE;
Product_Film_Handel_Run:=FALSE;
Process_1_Get_Finish:=FALSE;
Pressure_Fail_1:=FALSE;
Process_2_Can_Push:=FALSE;
Process_1_Push_Finish:=FALSE;
Process_1_Push_Finish_Sure:=FALSE;
Can_Move_Film:=FALSE;
Feed_1_Finish:=FALSE;
Y0_3:=FALSE;
bak_step:=0;
step:=0;
END_IF
END_PROGRAM

(* POU Run_Main_Folder/Right_Translation, ST *)
PROGRAM Right_Translation
VAR
	step: INT;
	bak_step:INT;
	rt_hold: R_TRIG;
	UP1: R_TRIG;
	T1:TON;
END_VAR

VAR_INPUT
	bstart1: BOOL;
	bhold1: BOOL;
	breset1: BOOL;


END_VAR
(*右平移程序流程*)

UP1(CLK:=Right_Translation_Run , Q=> );

CASE step OF
0:
 IF UP1.Q THEN
step:=1;
END_IF

1:
IF pan_have_liao2 THEN
	step:=30;
ELSE
step:=10;
END_IF

10:
D2:=A2_W1;(*右---等待放料工位*)
Axis2_MoveAbsolute:=TRUE;
IF Axis2_Abs_Function.Done THEN
Process_4_Can_Push:=TRUE; (*告知滚压可以放料*)
Axis2_MoveAbsolute:=FALSE;
step:=20;
END_IF;

20:
IF Process_3_Set_Finish THEN(*等待关押设备送料完成信号*)
	Process_3_Set_Finish:=FALSE;
	Y0_14:=TRUE;
	Y0_1:=TRUE;
	pan_have_liao2:=TRUE;
Get_Robort_simo_Finish:=FALSE;
	step:=30;
END_IF

30:(*此时载盘有料*)
D2:=A2_P1;
Axis2_MoveAbsolute:=TRUE;
IF Axis2_Abs_Function.Done THEN
Axis2_MoveAbsolute:=FALSE;
(*到位拍照*)
Flag_RightStage_Cam_Pos1_Ready:=TRUE;
step:=32;
END_IF

32:
IF Flag_RightStage_Cam_Pos1_Finish=TRUE THEN
	Flag_RightStage_Cam_Pos1_Ready:=FALSE;
	Flag_RightStage_Cam_Pos1_Finish:=FALSE;
	step:=34;
END_IF

34:
D2:=A2_P2;
Axis2_MoveAbsolute:=TRUE;
IF Axis2_Abs_Function.Done THEN
Axis2_MoveAbsolute:=FALSE;
Flag_RightStage_Cam_Pos2_Ready:=TRUE;
step:=36;
END_IF

36:
IF Flag_RightStage_Cam_Pos2_Finish=TRUE THEN
	Flag_RightStage_Cam_Pos2_Ready:=FALSE;
	Flag_RightStage_Cam_Pos2_Finish:=FALSE;
	step:=38;
END_IF

38:
D2:=A2_P3;
Axis2_MoveAbsolute:=TRUE;
IF Axis2_Abs_Function.Done THEN
Axis2_MoveAbsolute:=FALSE;
Flag_RightStage_RemoveLiner_Ready:=TRUE;
step:=40;
END_IF

40:
IF Flag_RightStage_Robot_RemoveLiner_Ready=TRUE THEN
	Flag_RightStage_RemoveLiner_Ready:=FALSE;
	Flag_RightStage_Robot_RemoveLiner_Ready:=FALSE;
	step:=42;
END_IF

42:
D2:=A2_P4;
Axis2_MoveAbsolute:=TRUE;
IF Axis2_Abs_Function.Done THEN
Axis2_MoveAbsolute:=FALSE;
Flag_RightStage_RemoveLinered_Ready:=TRUE;
step:=44;
END_IF

44:
IF Flag_RightStage_Robot_RemoveLinered_Ready THEN
	Flag_RightStage_RemoveLinered_Ready:=FALSE;
	Flag_RightStage_Robot_RemoveLinered_Ready:=FALSE;
	step:=46;
END_IF

46:
D2:=A2_P5;
Axis2_MoveAbsolute:=TRUE;
IF Axis2_Abs_Function.Done THEN
	Axis2_MoveAbsolute:=FALSE;
	Flag_Barcode_Can_Fit:=TRUE;
	step:=48;
END_IF

48:
IF Flag_Barcode_Fit_Finish=TRUE THEN
	Flag_Barcode_Fit_Finish:=FALSE;
	step:=50;
END_IF

50:
D2:=A2_P6;
Axis2_MoveAbsolute:=TRUE;
IF Axis2_Abs_Function.Done THEN
	Axis2_MoveAbsolute:=FALSE;
	Flag_RightStage_Cam_Brd1_Ready:=TRUE;
	step:=52;
END_IF

52:
IF Flag_RightStage_Cam_Brd1_Finish THEN
	Flag_RightStage_Cam_Brd1_Ready:=FALSE;
	step:=54;
END_IF

54:
D2:=A2_P7;
Axis2_MoveAbsolute:=TRUE;
IF Axis2_Abs_Function.Done THEN
	Axis2_MoveAbsolute:=FALSE;
	Flag_RightStage_Cam_Brd2_Ready:=TRUE;
	step:=56;
END_IF

56:
IF Flag_RightStage_Cam_Brd2_Finish THEN
	Flag_RightStage_Cam_Brd2_Ready:=FALSE;
	step:=58;
END_IF

58:
D2:=A2_P8;
Axis2_MoveAbsolute:=TRUE;
IF Axis2_Abs_Function.Done THEN
	Axis2_MoveAbsolute:=FALSE;
	Flag_RightStage_Cam_Brd3_Ready:=TRUE;
	step:=60;
END_IF

60:
IF Flag_RightStage_Cam_Brd3_Finish THEN
	Flag_RightStage_Cam_Brd3_Ready:=FALSE;
	step:=62;
END_IF

62:
D2:=A2_P9;
Axis2_MoveAbsolute:=TRUE;
IF Axis2_Abs_Function.Done THEN
	Axis2_MoveAbsolute:=FALSE;
	Flag_RightStage_Cam_Brd4_Ready:=TRUE;
	step:=64;
END_IF

64:
IF Flag_RightStage_Cam_Brd4_Finish THEN
	Flag_RightStage_Cam_Brd4_Ready:=FALSE;
	step:=66;
END_IF

66:
D2:=A2_P10;
Axis2_MoveAbsolute:=TRUE;
IF Axis2_Abs_Function.Done THEN
	Axis2_MoveAbsolute:=FALSE;
	Y1_11:=TRUE;(*松吸嘴*)
	Y0_14:=FALSE;
	Y0_1:=FALSE;

	Flag_RightStage_WaitCatch_Ready:=TRUE;
	step:=68;
END_IF

68:
IF Flag_RightStage_WaitCatch_Ready THEN
	Flag_RightStage_WaitCatch_Ready:=FALSE;
	step:=70;
END_IF

70:
IF Flag_RightStage_WaitCatch_Finish=TRUE THEN
	Y1_11:=FALSE;
	Flag_RightStage_WaitCatch_Finish:=FALSE;
	pan_have_liao2:=FALSE;
	Button_Ad:=FALSE;
	step:=1;
END_IF




300:
    IF bstart1   AND NOT Total_Axis_Error AND NOT total_pausestatus  THEN
	step:=bak_step;
END_IF;
END_CASE

T1(IN:=Y1_11 , PT:=t#4s , Q=> , ET=> );
IF T1.Q   THEN
Y1_11:=FALSE;
END_IF

rt_hold(CLK:=( Total_Axis_Error OR  bhold1) , Q=> ); (*暂停状态*)
IF step<>0 AND step<>300   AND  rt_hold.Q THEN
     bak_step:=step;
     step:=300;
END_IF

IF Total_Emergency THEN
	Y1_11:=FALSE;
	Right_Translation_Run:=FALSE;

	Flag_RightStage_Cam_Pos1_Ready:=FALSE;
	Flag_RightStage_Cam_Pos2_Ready:=FALSE;

	Flag_RightStage_Cam_Brd1_Ready:=FALSE;
	Flag_RightStage_Cam_Brd2_Ready:=FALSE;
	Flag_RightStage_Cam_Brd3_Ready:=FALSE;
	Flag_RightStage_Cam_Brd4_Ready:=FALSE;

	Flag_RightStage_Cam_Pos1_Finish:=FALSE;
	Flag_RightStage_Cam_Pos2_Finish:=FALSE;

	Flag_RightStage_Cam_Brd1_Finish:=FALSE;
	Flag_RightStage_Cam_Brd2_Finish:=FALSE;
	Flag_RightStage_Cam_Brd3_Finish:=FALSE;
	Flag_RightStage_Cam_Brd4_Finish:=FALSE;

	Flag_RightStage_RemoveLiner_Ready:=FALSE;
	Flag_RightStage_Robot_RemoveLiner_Ready:=FALSE;
	Flag_RightStage_RemoveLinered_Ready:=FALSE;
	Flag_RightStage_Robot_RemoveLinered_Ready:=FALSE;

	Flag_RightStage_WaitCatch_Ready:=FALSE;
	Flag_RightStage_WaitCatch_Finish:=FALSE;

	Y0_14:=FALSE;
	Y0_1:=FALSE;
	Y0_12:=FALSE;
	pan_have_liao2:=FALSE;
	Process_4_Can_Push:=FALSE; (*告知滚压可以放料*)
	Process_3_Set_Finish:=FALSE;
	bak_step:=0;
	step:=0;
END_IF
END_PROGRAM

(* POU Run_Main_Folder/Rolling_Part, ST *)
PROGRAM Rolling_Part
VAR
	step: INT;
	bak_step:INT;
	rt_hold: R_TRIG;
	UP1: R_TRIG;
	T1: TON;
	T2:TON;
	T3:TON;
	T6: TON;

END_VAR

VAR_INPUT
	bstart1: BOOL;
	bhold1: BOOL;
	breset1: BOOL;

END_VAR
(*滚压部分程序*)

UP1(CLK:=Rolling_Part_Run , Q=> );

CASE step OF
0:
 IF UP1.Q THEN
step:=10;
END_IF

10:(*滚压部分开始动作*)
(*判断机械手是否放好料---------放好之后，进行滚压动作，询问右移载是否可以送料，可送料之后，给出料，同时，发出，给料完成信号*)
IF rolling_have_liao THEN
	step:=100;
ELSE
step:=20;
END_IF

20:(*无料的操作*)
D10:=A10_W2;
Axis10_MoveAbsolute:=TRUE;
IF Axis10_Abs_Function.Done THEN
Axis10_MoveAbsolute:=FALSE;
Process_3_Can_Push:=TRUE;

step:=29;
END_IF

29:(*机械手2放下后，告知可以开吸嘴*)
IF Wait_Robot_Push THEN
Wait_Robot_Push:=FALSE;
Y0_12:=TRUE;(*滚压平台*)
step:=31;
END_IF

31:
	IF Empty_Pro THEN

	step:=30;
	ELSE
Y0_12:=TRUE;(*滚压平台*)
	step:=30;
END_IF


30:(*等待机械手2.放料*)
IF Robot2_Push_Finish THEN
Rolling_Number:=0;
rolling_have_liao:=TRUE;
Process_3_Can_Push:=FALSE;
Robot2_Push_Finish:=FALSE;
Y0_10:=TRUE;(*推入气缸*)
step:=50;
END_IF


50:
IF X2_16 THEN
(*Y0_9:=TRUE;*)
Y0_11:=TRUE;
step:=51;
END_IF

60:
V23:=A23PRoll;(*滚压Z轴滚压位*)
Axis23_MoveAbsolute:=TRUE;
IF Axis23_Abs_Function.Done THEN
	Axis23_MoveAbsolute:=FALSE;
	step:=70;
END_IF


(*60:
IF X3_2  THEN(*压合气缸到位，等待滚压*)
step:=70;
END_IF*)

70:
D10_1:=A10_W1;(*出去位置*)(*滚压低速*)
Axis10_MoveAbsolute1:=TRUE;
IF Axis10_Abs_Function1.Done THEN
Axis10_MoveAbsolute1:=FALSE;

Y0_11:=FALSE;
step:=78;
END_IF

78:
V23:=A23PInit;(*滚压Z轴滚压位*)
Axis23_MoveAbsolute:=TRUE;
IF Axis23_Abs_Function.Done THEN
	Axis23_MoveAbsolute:=FALSE;
	step:=80;
END_IF

80:
D10:=A10_W2;
Axis10_MoveAbsolute:=TRUE;
IF Axis10_Abs_Function.Done THEN
Axis10_MoveAbsolute:=FALSE;
Rolling_Number:=Rolling_Number+1;
step:=90;
END_IF

90:
IF Rolling_Number>=Set_Rolling_Number THEN
Rolling_Number:=0;

Y0_9:=FALSE;
step:=100;(*次数满足，跳转*)
ELSE
step:=50;
END_IF

100:
IF X3_3 THEN
Y0_10:=FALSE;
step:=110;
END_IF

110:
IF X3_1 THEN
step:=120;
END_IF

120:(*滚压回到安全位置------询问是否可以扣料*)
IF Process_4_Can_Push THEN
Process_4_Can_Push:=FALSE;
Y0_13:=TRUE;(*翻转动作开始动作*)
step:=130;
END_IF

130:
IF X3_4 THEN

step:=131;
END_IF

131:
IF Empty_Pro THEN
step:=139;
ELSE
Y0_14:=TRUE;(*右真空吸开始吸取*)
Y0_1:=TRUE;
step:=139;
END_IF


139:
T6(IN:=TRUE , PT:=t#0.4s , Q=> , ET=> );
IF T6.Q   THEN
T6(IN:=FALSE, PT:=t#0.4S , Q=> , ET=> );
Y0_12:=FALSE;
step:=140;
END_IF

140:
T2(IN:=TRUE , PT:=t#0.4s , Q=> , ET=> );
   IF T2.Q   THEN
T2(IN:=FALSE, PT:=t#0.4S , Q=> , ET=> );
rolling_have_liao:=FALSE;
Y0_13:=FALSE;
step:=150;
END_IF

150:
IF X3_5 THEN(*翻转结构�--------完成------告知机械手*)
	T3(IN:=TRUE , PT:=t#0.4s , Q=> , ET=> );
	 IF T3.Q   THEN
		T3(IN:=FALSE, PT:=t#0.4S , Q=> , ET=> );
		Process_3_Set_Finish:=TRUE;
		step:=10;
	END_IF
END_IF


300:
    IF bstart1   AND NOT Total_Axis_Error AND NOT total_pausestatus  THEN
	step:=bak_step;
END_IF;
END_CASE

rt_hold(CLK:=( Total_Axis_Error OR  bhold1) , Q=> ); (*暂停状态*)
IF step<>0 AND step<>300   AND  rt_hold.Q THEN
     bak_step:=step;
     step:=300;
END_IF



IF Total_Emergency THEN
Rolling_Part_Run:=FALSE;
Process_3_Set_Finish:=FALSE;
Process_3_Can_Push:=FALSE;

rolling_have_liao:=FALSE;
Process_3_Can_Push:=FALSE;
Wait_Robot_Push:=FALSE;
Robot2_Push_Finish:=FALSE;
Rolling_Number:=0;
Process_4_Can_Push:=FALSE;
Process_3_Set_Finish:=FALSE;


bak_step:=0;
step:=0;
END_IF
END_PROGRAM

(* POU Run_Main_Folder/Left_FPC_Feed/Left_Carry, ST *)
PROGRAM Left_Carry
VAR
	step: INT;
	bak_step:INT;
	rt_hold: R_TRIG;
	UP1: R_TRIG;
	T1: TON;

	T2: TON;

	T8: TON;
END_VAR

VAR_INPUT
	bstart1: BOOL;
	bhold1: BOOL;
	breset1: BOOL;

END_VAR
(*fpc气缸移载程序。。。。*)


UP1(CLK:=Left_Carry_Run , Q=> );

CASE step OF
0:
 IF UP1.Q THEN
step:=10;
END_IF

(*等待机械手取完信号，当移载完成之后，给左可上升信号，放下料之后给出，左可下降信号*)
10:
IF Left_hand_have THEN
(*手上有料，则直接放料位置*)
step:=80;
ELSE
step:=20;
END_IF


20:(*判断是否机械手取空*)
IF  Left_Can_Move THEN
Left_Can_Move:=FALSE;(*等待到可平移信号*)
step:=30;
Y0_6:=TRUE;(*推杆气缸侗族*)
END_IF

30:
IF X2_10 THEN
Y0_7:=TRUE;
step:=40;
END_IF

40:
IF X2_12 THEN
Y0_8:=TRUE;
step:=50;
END_IF

50:
T1(IN:=TRUE , PT:=t#0.8s , Q=> , ET=> );
   IF T1.Q AND NOT Total_Pause  THEN
T1(IN:=FALSE, PT:=t#0.8S , Q=> , ET=> );
Y0_7:=FALSE;
step:=60;
END_IF

60:
IF X2_13 THEN(*气缸上抬到位*)
step:=68;
END_IF

68:
T8(IN:=TRUE , PT:=t#1s , Q=> , ET=> );
   IF T8.Q AND NOT Total_Pause  THEN
T8(IN:=FALSE, PT:=t#1S , Q=> , ET=> );
step:=70;
END_IF


70:(*判断是否吸取成功*)
IF X2_14 THEN
Y0_6:=FALSE;
Y1_9:=TRUE;(*上料完成，扣紧托盘*)
step:=80;
(*吸取成功*)
ELSE
Pressure_Left_Fail:=TRUE;
step:=30;(*重复吸取-----等待成功*)
END_IF

80:(*成功之后----给出可以上顶*)
IF X2_11 THEN
Left_Move_Finish:=TRUE;
step:=90;
END_IF

90:(*上方询问是否可放*)
IF zuo_down_Finish THEN
zuo_down_Finish:=FALSE;
Y0_7:=TRUE;
step:=100;
END_IF

100:
IF X2_12 THEN
Y0_8:=FALSE;
step:=110;
END_IF

110:
T2(IN:=TRUE , PT:=t#0.8s , Q=> , ET=> );
   IF T2.Q AND NOT Total_Pause  THEN
T2(IN:=FALSE, PT:=t#0.8S , Q=> , ET=> );
Y0_7:=FALSE;
step:=120;
END_IF

120:
IF X2_13 THEN
zuo_ke_jiang:=TRUE;
step:=10;
END_IF

300:
    IF bstart1   AND NOT Total_Axis_Error AND NOT total_pausestatus  THEN
	step:=bak_step;
END_IF;
END_CASE


rt_hold(CLK:=( Total_Axis_Error OR  bhold1) , Q=> ); (*暂停状态*)
IF step<>0 AND step<>300   AND  rt_hold.Q THEN
     bak_step:=step;
     step:=300;
END_IF

IF Total_Emergency THEN
y0_8:=FALSE;
Left_Carry_Run:=FALSE;
zuo_ke_jiang:=FALSE;
Left_Move_Finish:=FALSE;
bak_step:=0;
step:=0;
END_IF
END_PROGRAM

(* POU Run_Main_Folder/Liftin_Feed_1, ST *)
PROGRAM Liftin_Feed_1
VAR
	step: INT;
	bak_step:INT;
	rt_hold: R_TRIG;
	UP1: R_TRIG;
	T1: TON;
	T2:TON;
	T3:TON;

	T5: TON;
END_VAR

VAR_INPUT
	bstart1: BOOL;
	bhold1: BOOL;
	breset1: BOOL;

END_VAR
(*FG上料程序*)
(*上料上升，开始动作，当感应到传感器，停止运行，告知，上料完成，，，，同时接收取完信号，当取完信号右了
此时，循环上升，？？？？？何时检测极限信号，同时下降之后报警报警不暂停，等待上料按钮---------*)

UP1(CLK:=Liftin_Feed_1_Run , Q=> );

CASE step OF

0:
 IF UP1.Q
THEN step:=1;
END_IF

1:
IF (X100_6  AND X101_11)OR (X100_7 AND X101_12) THEN
	step:=10;
	(*在左边或者右边*)
	(*上升运行*)
ELSIF( X101_11 AND NOT  X100_6 ) OR ( X101_12  AND NOT X100_7) THEN
	step:=2;
	(*错位*)
ELSE
	FGFeed1Empty:=TRUE;
	FGFeed2Empty:=TRUE;
	step:=60;
END_IF

2:
(*错位*)
IF axis3.NcToPlc.ActPos <= 5
THEN Y100_2:= NOT Y100_2; step:=3;(*取反气缸，延时2秒*)
ELSE step:=50;(*碰到极限，此时料取完,回到初始位置*)
END_IF

3:
T5(IN:=TRUE , PT:=t#2s , Q=> , ET=> );
IF T5.Q   THEN
	T5(IN:=FALSE, PT:=t#2S , Q=> , ET=> );
	step:=1;
END_IF

10:(*上升运行*)
Axis3_PTF_2:=TRUE;
Axis3_Halt:=FALSE;
IF (((X2_1 AND x100_6)OR(x100_4 AND x100_7)) AND  X0_1) OR Empty_Pro THEN(*碰到光纤，同时没有碰到极限，此时上料ok*)
	Axis3_PTF_2:=FALSE;
	IF NOT Discharge_Button THEN
		Feed_1_Finish:=TRUE;
	END_IF

	Axis3_Halt:=TRUE;
	step:=20;
END_IF
IF NOT  X0_1 THEN(*碰到极限，此时表示料空*)
	Axis3_PTF_2:=FALSE;
	Axis3_Halt:=TRUE;
	IF x100_6 THEN
		FGFeed1Empty:=TRUE;
	END_IF
	IF x100_7 THEN
		FGFeed2Empty:=TRUE;
	END_IF

	IF  Discharge_Button THEN
	Discharge_Button:=FALSE;
	END_IF
step:=50;
END_IF

20:
Axis3_Halt:=FALSE;
(*表示上料成功,等待取完信号*)
IF Process_1_Get_Finish AND NOT Discharge_Button  THEN

T3(IN:=TRUE , PT:=t#0.1s , Q=> , ET=> );
IF T3.Q AND NOT Total_Pause  THEN
	T3(IN:=FALSE, PT:=t#0.1S , Q=> , ET=> );
	Process_1_Get_Finish:=FALSE;
	step:=10;
END_IF

END_IF
IF Discharge_Button THEN
Discharge_Button:=FALSE;
Feed_1_Finish:=FALSE;
step:=50;
END_IF

50:(*碰到极限，此时料取完,回到初始位置*)
Axis3_Halt:=FALSE;
D3:=D300;
Axis3_MoveAbsolute:=TRUE;
IF Axis3_Abs_Function.Done THEN
Axis3_MoveAbsolute:=FALSE;
Feed_1_Nome_Alam:=TRUE;(*不暂停，只提示*)
step:=60;
END_IF

60:(*回到初始位置，提示料空*)
IF NOT FGFeed1Empty OR NOT FGFeed2Empty THEN
	step:=2;
END_IF
IF UP_Button AND NOT Total_Pause AND X101_11  THEN
FGFeed1Empty:=FALSE;
FGFeed2Empty:=FALSE;
Feed_1_Nome_Alam:=FALSE;
UP_Button:=FALSE;
step:=1;
END_IF

300:
IF bstart1   AND NOT Total_Axis_Error AND NOT total_pausestatus THEN
	step:=bak_step;
END_IF;
END_CASE


rt_hold(CLK:=( Total_Axis_Error OR  bhold1) , Q=> ); (*暂停状态*)
IF step<>0 AND step<>300   AND  rt_hold.Q THEN
     bak_step:=step;
	Axis3_Halt:=TRUE;
     step:=300;
END_IF

IF UP_Button THEN
	IF  FGFeed1Empty AND NOT  FGFeed2Empty
	THEN FGFeed1Empty:=FALSE;
	END_IF
	
	IF NOT  FGFeed1Empty AND   FGFeed2Empty
	THEN FGFeed2Empty:=FALSE;
	END_IF
	UP_Button:=FALSE;
END_IF

IF Total_Emergency THEN
Liftin_Feed_1_Run:=FALSE;
Feed_1_Finish:=FALSE;
Feed_1_Nome_Alam:=FALSE;
Discharge_Button:=FALSE;
Empty_Pro:=FALSE;

bak_step:=0;
step:=0;
END_IF

(*随时可以不做料的操作*)
IF Feed1_Button AND step=20 AND NOT Total_Pause THEN
Feed1_Button:=FALSE;
Feed_1_Finish:=FALSE;
step:=50;
ELSE
Feed1_Button:=FALSE;
END_IF
END_PROGRAM

(* POU Run_Main_Folder/Left_FPC_Feed/Liftin_Feed_Left_1, ST *)
PROGRAM Liftin_Feed_Left_1
VAR

	step: INT;
	flag_nostop:BOOL;
	bak_step:INT;
	rt_hold: R_TRIG;
	UP1: R_TRIG;
	T1: TON;
	T2:TON;

	CurHeight:LREAL;
END_VAR

VAR_INPUT
	bstart1: BOOL;
	bhold1: BOOL;
	breset1: BOOL;

END_VAR
(*FPC上料程序*)

(*上升供料电机流程*)

UP1(CLK:=Liftin_Feed_Left_1_Run OR Specila_Feed_FPC , Q=> );

CASE step OF
0:
 IF UP1.Q THEN
step:=10;
END_IF

10:(*上升运行*)
Feed_Left_None_Alam:=FALSE;(*不暂停，只提示*)
flag_nostop:=FALSE;
Flag_FPC_brd_Err:=FALSE;
Y1_9:=TRUE;(*上料完成，扣紧托盘*)
Axis6_PTF_2:=TRUE;
IF X2_2 AND  X0_10 THEN(*碰到光纤，同时没有碰到极限，此时上料ok*)
	Axis6_PTF_2:=FALSE;
	Axis6_Halt:=TRUE;
	IF axis6.NcToPlc.ActPos>253.5 THEN
		step:=11;
	ELSE
		Feed_2_Finish:=TRUE;
		step:=20;
	END_IF

END_IF
IF NOT  X0_10 THEN(*碰到极限，此时表示料空*)
Axis6_PTF_2:=FALSE;
Axis6_Halt:=TRUE;
step:=50;
END_IF

11:
Axis6_Halt:=FALSE;
D6:=254;(*先抬高一点，然后置位平托气缸253.5*)
Axis6_MoveAbsolute:=TRUE;
IF Axis6_Abs_Function.Done THEN
Axis6_MoveAbsolute:=FALSE;
Feed_2_Finish:=TRUE;
step:=12;
END_IF

12:
Y100_9:=TRUE;
Feed_2_Finish:=TRUE;
Axis6_PTF_2:=FALSE;
Axis6_Halt:=TRUE;
flag_nostop:=TRUE;
step:=50;



20:
Axis6_Halt:=FALSE;
(*表示上料成功,等待取完信号*)
IF Get_Robot1_Tray_Empty  THEN
Y1_9:=FALSE;(*取料完成，松开*)
Feed_2_Finish:=FALSE;
Left_Can_Move:=TRUE;
Get_Robot1_Tray_Empty:=FALSE;(*上料完成，机械手取空*)
step:=30;
END_IF

IF Flag_FPC_brd_Err THEN
Y1_9:=FALSE;(*取料完成，松开*)
Feed_2_Finish:=FALSE;
step:=21;
END_IF

21:(*最后一盘扫码失败，必须拿掉，否则你懂得*)
IF NOT Flag_FPC_brd_Err THEN
IF flag_nostop=TRUE THEN
	Y100_9:=FALSE;
	flag_nostop:=FALSE;
	step:=60;
ELSE
	step:=10;
END_IF
END_IF

30:(*等待平移完成，才可以上升*)
IF Left_Move_Finish THEN
Left_Move_Finish:=FALSE;
IF flag_nostop=TRUE THEN
	Y100_9:=FALSE;
	flag_nostop:=FALSE;
	step:=60;
ELSE
	step:=10;
END_IF
END_IF

50:(*碰到极限，此时料取完,回到初始位置*)
Axis6_Halt:=FALSE;
D6:=D600;
Axis6_MoveAbsolute:=TRUE;
IF Axis6_Abs_Function.Done THEN
Axis6_MoveAbsolute:=FALSE;
Feed_Left_None_Alam:=TRUE;(*不暂停，只提示*)
	IF flag_nostop=TRUE THEN
		step:=20;
	ELSE
		step:=60;
	END_IF

END_IF

60:(*回到初始位置，提示料空*)
IF Left_UP_Button AND NOT Total_Pause THEN
Left_UP_Button:=FALSE;
step:=10;
END_IF

300:
    IF bstart1   AND NOT Total_Axis_Error AND NOT total_pausestatus  THEN
	step:=bak_step;
END_IF;
END_CASE



rt_hold(CLK:=( Total_Axis_Error OR  bhold1) , Q=> ); (*暂停状态*)
IF step<>0 AND step<>300   AND  rt_hold.Q THEN
     bak_step:=step;
     step:=300;
END_IF


IF Left_UP_Button THEN
Left_UP_Button:=FALSE;
END_IF

IF Total_Emergency OR Specila_Feed_FPC_OFF  THEN
Specila_Feed_FPC:=FALSE;
Liftin_Feed_Left_1_Run:=FALSE;
Feed_Left_None_Alam:=FALSE;
bak_step:=0;
Feed_2_Finish:=FALSE;
Y1_9:=FALSE;


step:=0;
END_IF



(*随时可以不做料的操作*)
IF Feed_Left_Button1 AND step=20 AND NOT Total_Pause THEN
Feed_Left_Button1:=FALSE;
Feed_2_Finish:=FALSE;
step:=50;
ELSE
Feed_Left_Button1:=FALSE;
END_IF
END_PROGRAM

(* POU Run_Main_Folder/Left_FPC_Feed/Liftin_Feed_Left_2, ST *)
PROGRAM Liftin_Feed_Left_2
VAR

	step: INT;
	bak_step:INT;
	rt_hold: R_TRIG;
	UP1: R_TRIG;
	DOWN1: F_TRIG;

	T1: TON;
	T2:TON;
	T3:TON;
	flag_nostop:BOOL;
END_VAR

VAR_INPUT
	bstart1: BOOL;
	bhold1: BOOL;
	breset1: BOOL;

END_VAR
(*fpc空盘下料程序*)

(*左下降，初始化，回原点到初始位置，，，启动之后，先往上走，到初始位置(第一次回原点使用)  ，接收到送料完成可下降信号，则
开始下降，等现将结束，告知，可放料*)

UP1(CLK:=Liftin_Feed_Left_2_Run , Q=> );

CASE step OF
0:
 IF UP1.Q THEN
step:=1;
END_IF

1:
(*初始化之后位置在下面的初始位置*)
Axis7_PTF_2:=TRUE;
IF X2_3 AND X0_13 THEN(*碰到光纤说明此时有料，则停止，等待跳转到20等到下降到光纤下降沿*)
Axis7_PTF_2:=FALSE;
Axis7_Halt:=TRUE;
step:=20;
END_IF
IF NOT X0_13 THEN(*上极限的时候，说明此时物料，跳转到60，回到上初始位置*)
Axis7_PTF_2:=FALSE;
Axis7_Halt:=TRUE;
step:=60;(*撞到极限，此时需要回到上面的初始位置*)
END_IF

10:
(*初始化的时候写，回原点之后，向上跑知道碰到光纤，或者极限的时候，到极限回到初始位置，碰到光纤，停止，翻转到极限停止位置*)

(*到初始位置，等待放料，当光纤感应到，同时，接收到，可下降信号的时候，开始下降，当感应不到光纤，则停止*)
IF zuo_ke_jiang AND X2_3 THEN
zuo_ke_jiang:=FALSE;
	step:=20;
END_IF

20:
Axis7_Halt:=FALSE;
(*接收到可降信号，开始下降，到传感器下降沿停止下降，等待*)
Axis7_PTF:=TRUE;
DOWN1(CLK:=X2_3 , Q=> );
IF DOWN1.Q AND NOT   (axis7.NcToPlc.ActPos<=50) THEN (*未碰到原点，此时，光纤下降沿*)
Axis7_PTF:=FALSE;
zuo_down_Finish:=TRUE;
Axis7_Halt:=TRUE;
step:=30;
END_IF
IF (axis7.NcToPlc.ActPos<=60)    THEN(*碰到原点，此时表示料空X0_14*)
Y100_10:=TRUE;
zuo_down_Finish:=TRUE;

Axis7_PTF:=FALSE;
Axis7_Halt:=TRUE;
step:=400;
END_IF

30:(*停止，给出下降完成信号，等待放料循环*)
Axis7_Halt:=FALSE;
T3(IN:=TRUE , PT:=t#0.2s , Q=> , ET=> );
IF T3.Q AND NOT Total_Pause  THEN
	T3(IN:=FALSE, PT:=t#0.2S , Q=> , ET=> );
	zuo_down_Finish:=TRUE;
	step:=10;
END_IF

400:(*碰到原点，此时，回到下初始位置，给出料满提示*)
Axis7_Halt:=FALSE;
D7:=D700;
Axis7_MoveAbsolute:=TRUE;
IF Axis7_Abs_Function.Done THEN
Axis7_MoveAbsolute:=FALSE;
Feed_Left_Full_Alam:=TRUE;(*不暂停，只提示*)
step:=50;
END_IF

50:(*碰到下极限，给出缺料提示*)
Axis7_Halt:=FALSE;
IF Left_Down_Button AND NOT Total_Pause THEN
	Left_Down_Button:=FALSE;
	Feed_Left_Full_Alam:=FALSE;
	step:=1;(*确认拿走料之后，运动到初始位置*)
END_IF

60:(*回到初始位置*)
Axis7_Halt:=FALSE;
D7:=D710;
Axis7_MoveAbsolute:=TRUE;
IF Axis7_Abs_Function.Done THEN
Axis7_MoveAbsolute:=FALSE;
zuo_down_Finish:=TRUE;(*左下降完成信号*)
step:=10;
END_IF

300:
    IF bstart1   AND NOT Total_Axis_Error AND NOT total_pausestatus THEN
	step:=bak_step;
END_IF;
END_CASE

rt_hold(CLK:=( Total_Axis_Error OR  bhold1) , Q=> ); (*暂停状态*)
IF step<>0 AND step<>300   AND  rt_hold.Q THEN
     bak_step:=step;
     step:=300;
END_IF


IF Total_Emergency THEN
Liftin_Feed_Left_2_Run:=FALSE;
zuo_down_Finish:=FALSE;
Feed_Left_Full_Alam:=FALSE;

bak_step:=0;
step:=0;
END_IF

(*随时可以不做料的操作*)
IF Feed_Left_Button2 AND step=10 AND NOT Total_Pause THEN
Feed_Left_Button2:=FALSE;
zuo_down_Finish:=FALSE;
step:=400;
ELSE
Feed_Left_Button2:=FALSE;
END_IF
END_PROGRAM

(* POU Run_Main_Folder/Left_Translation/New_Table_1, ST *)
PROGRAM New_Table_1
VAR
	step: INT;
	bak_step:INT;
	rt_hold: R_TRIG;
	UP1: R_TRIG;
	Run_Time:BOOL;
	T1:TON;
	Run_Time_Lreal: TIME;
	T3:TON;




	T2: TON;

END_VAR

VAR_INPUT
	bstart1: BOOL;
	bhold1: BOOL;
	breset1: BOOL;

END_VAR
(*滑台1程序*)


UP1(CLK:=Left_Translation_Run_1 , Q=> );


(*首先上料-------------------此时位置*)
CASE step OF
0:
 IF UP1.Q THEN
step:=10;
END_IF

10:(*判断是否有料*)
IF Tray1_Have THEN
step:=60;
ELSE
step:=20;
END_IF

20:
D1:=A1_W1;(*左等待放料工位*)
Axis1_MoveAbsolute:=TRUE;
IF Axis1_Abs_Function.Done THEN
Process_2_Can_Push1:=TRUE;(*告知上料部分可以上料*)
Axis1_MoveAbsolute:=FALSE;
step:=30;
END_IF;

30:(*到位置之后，给出，可上料信号--------------等待上料完成信号----------上料完成后，等待真空吸完成*)
IF Process_1_Push_Finish THEN
Tray1_Have:=TRUE;
Process_1_Push_Finish:=FALSE;
step:=40;
END_IF

40:
T2(IN:=TRUE , PT:=t#0.5s , Q=> , ET=> );
   IF T2.Q AND NOT Total_Pause  THEN
T2(IN:=FALSE, PT:=t#0.5S , Q=> , ET=> );
Can_Move_Film:=TRUE;(*给出可撕膜信号*)
step:=50;
END_IF

50:(*给出可撕膜信号*)
IF Process_1_Push_Finish_Sure THEN
Process_1_Push_Finish_Sure:=FALSE;
step:=60;
END_IF

60:(*判断拍照位置1是否安全*)
IF Positive_Camera_Safe1 THEN
Positive_Camera_Safe1:=FALSE;(*拍照位置1被占据*)
step:=70;
END_IF

70:
D1:=A1_W2;(*拍照工位1*)
Axis1_MoveAbsolute:=TRUE;
IF Axis1_Abs_Function.Done THEN
Axis1_MoveAbsolute:=FALSE;
(*到位拍照*)
Camera_1_1_run:=TRUE;
step:=80;
END_IF

80:(*拍照工位1拍照结束-----等待*)
IF Camera_1_1_OK THEN
Camera_1_1_run:=FALSE;
Camera_1_1_OK:=FALSE;
step:=90;
END_IF
IF Camera1_NG THEN  (*拍照失败的处理，判断ng,此时需要给出结果，，，，，，，同时运动到工作位置*)
Camera_1_1_run:=FALSE;
Tray1_Have:=FALSE;
Camera1_NG:=FALSE;
Y0_5:=FALSE;
step:=2000;
END_IF



90:(*判断拍照位置2是否安全*)
IF Positive_Camera_Safe2 THEN
Positive_Camera_Safe2:=FALSE;
step:=100;
END_IF

100:(*移动到位置2*)
D1:=A1_W3; (*拍照工位2*)
Axis1_MoveAbsolute:=TRUE;
IF Axis1_Abs_Function.Done THEN
Axis1_MoveAbsolute:=FALSE;
(*到位拍照*)
Camera_1_2_run:=TRUE;
step:=110;
END_IF

110:
IF Camera_1_2_OK THEN
Camera_1_2_run:=FALSE;
Camera_1_2_OK:=FALSE;
step:=120;
END_IF
IF Camera1_NG THEN  (*拍照失败的处理，判断ng,此时需要给出结果，，，，，，，同时运动到工作位置*)
Camera_1_2_run:=FALSE;
Tray1_Have:=FALSE;
Camera1_NG:=FALSE;
Y0_5:=FALSE;
step:=2020;
END_IF

120:(*判断位置3是否安全*)
IF Positive_Camera_Safe3 THEN
Positive_Camera_Safe3:=FALSE;
step:=130;
END_IF

130:(*到工位3*)
D1:=A1_W4;(*拍照工位3*)
Axis1_MoveAbsolute:=TRUE;
IF Axis1_Abs_Function.Done THEN
Axis1_MoveAbsolute:=FALSE;
(*到位拍照*)
Camera_1_3_run:=TRUE;
step:=140;
END_IF

140:
IF Camera_1_3_OK THEN
Camera_1_3_run:=FALSE;
Camera_1_3_OK:=FALSE;
step:=150;
END_IF
IF Camera1_NG THEN  (*拍照失败的处理，判断ng,此时需要给出结果，，，，，，，同时运动到工作位置*)
Camera_1_3_run:=FALSE;
Tray1_Have:=FALSE;
Camera1_NG:=FALSE;
Y0_5:=FALSE;
step:=2050;
END_IF


150:(*拍照位置3判断是否安全----------*)
IF Positive_Camera_Safe4 THEN
Positive_Camera_Safe4:=FALSE;
step:=160;
END_IF

160:
D1:=A1_W5;(*拍照工位4*)
Axis1_MoveAbsolute:=TRUE;
IF Axis1_Abs_Function.Done THEN
Axis1_MoveAbsolute:=FALSE;
(*到位拍照*)
Positive1_Safe:=TRUE;

Camera_1_4_run:=TRUE;
step:=170;
END_IF

170:
IF Camera_1_4_OK THEN
Camera_1_4_run:=FALSE;
Camera_1_4_OK:=FALSE;
step:=180;
END_IF
IF Camera1_NG THEN  (*拍照失败的处理，判断ng,此时需要给出结果，，，，，，，同时运动到工作位置*)
Camera_1_4_run:=FALSE;
Tray1_Have:=FALSE;
Camera1_NG:=FALSE;
Y0_5:=FALSE;
step:=2070;
END_IF


180:(*判断工作位置1是否安全*)
IF Positive_Fit_Safe1 THEN
Positive_Fit_Safe1:=FALSE;
(*
HB_Fit_Finish_1:=FALSE;
HB_Fit_Finish_2:=FALSE;
HB_Fit_Finish_3:=FALSE;
HB_Fit_Finish_4:=FALSE;*)

step:=190;
END_IF

190:(*到工作位置1*)
D1:=A1_W6;(*工作位置工位1*)
Axis1_MoveAbsolute:=TRUE;
IF Axis1_Abs_Function.Done THEN

Positive_Camera_Safe1:=TRUE;(*工作位置1是给出拍照位置1安全安全位置-------------------------------------*)

Axis1_MoveAbsolute:=FALSE;
FG_Ready_1:=TRUE;
Process_2_Set_Finish1:=TRUE;(*给机械手可贴合信号*)


step:=200;
END_IF

200:(*到位等待贴合完成*)
IF HB_Fit_Finish_1 THEN
FG_Ready_1:=FALSE;
HB_Fit_Finish_1:=FALSE;
step:=210;
END_IF

210:(*工位1贴合完成-----询问工作位置2是否安全*)
IF Positive_Fit_Safe2 THEN
Positive_Fit_Safe2:=FALSE;
step:=220;
END_IF

220:(*位置安全------到贴合位置2*)
D1:=A1_W7;(*工作位置工位1*)
Axis1_MoveAbsolute:=TRUE;
IF Axis1_Abs_Function.Done THEN
Axis1_MoveAbsolute:=FALSE;

Positive_Camera_Safe2:=TRUE;(*工作位置1是给出拍照位置1安全安全位置-------------------------------------*)

FG_Ready_2:=TRUE;
step:=230;
END_IF

230:(*等待贴合完成信号*)
IF HB_Fit_Finish_2 THEN
FG_Ready_2:=FALSE;
HB_Fit_Finish_2:=FALSE;
step:=240;
END_IF

240:(*贴合完成------寻问位置3是否安全*)
IF Positive_Fit_Safe3 THEN
Positive_Fit_Safe3:=FALSE;
step:=250;
END_IF

250:(*位置安全------到贴合位置2*)
D1:=A1_W8;(*工作位置工位1*)
Axis1_MoveAbsolute:=TRUE;
IF Axis1_Abs_Function.Done THEN
Axis1_MoveAbsolute:=FALSE;

Positive_Camera_Safe3:=TRUE;(*工作位置1是给出拍照位置1安全安全位置-------------------------------------*)

FG_Ready_3:=TRUE;
step:=260;
END_IF

260:(*等待贴合完成信号*)
IF HB_Fit_Finish_3 THEN
FG_Ready_3:=FALSE;
HB_Fit_Finish_3:=FALSE;
step:=270;
END_IF

270:(*位置3贴合完成，询问位置4是否安全*)
IF Positive_Fit_Safe4 THEN
Positive_Fit_Safe4:=FALSE;
step:=280;
END_IF

280:(*位置安全------到贴合位置2*)
D1:=A1_W9;(*工作位置工位1*)
Axis1_MoveAbsolute:=TRUE;
IF Axis1_Abs_Function.Done THEN
Axis1_MoveAbsolute:=FALSE;

Positive_Camera_Safe4:=TRUE;(*工作位置1是给出拍照位置1安全安全位置-------------------------------------*)

FG_Ready_4:=TRUE;
step:=290;
END_IF

290:(*等待贴合完成信号*)
IF HB_Fit_Finish_4 THEN
FG_Ready_4:=FALSE;
Process_2_Set_Finish1:=FALSE;(*给机械手可贴合信号*)
HB_Fit_Finish_4:=FALSE;
step:=300;
END_IF

300:(*位置4贴合完成--------------寻味位置*)
IF Positive2_Safe THEN
	Positive2_Safe:=FALSE;
	step:=310;
END_IF

310:(*位置到位后，等待，送吸嘴*)
IF Wait_Robort2_Touch_Finish  THEN
Wait_Robort2_Touch_Finish:=FALSE;
Y0_5:=FALSE;
step:=320;
END_IF

320:(*延时等待--------------*)
T3(IN:=TRUE , PT:=t#1s , Q=> , ET=> );
   IF T3.Q AND NOT Total_Pause  THEN
T3(IN:=FALSE, PT:=t#1S , Q=> , ET=> );
step:=340;
END_IF

340:(*延时结束，等到最终完成信号*)
IF Get_Robot1_Get_Finish THEN
Tray1_Have:=FALSE;
Get_Robot1_Get_Finish:=FALSE;
step:=350;
END_IF

350:(*当完成最终取走的信号-------询问位置3是否安全*)
IF Positive3_Safe THEN
	Positive3_Safe:=FALSE;
	Y1_6:=TRUE;
	step:=360;
END_IF

360:
IF X4_12 THEN
Positive2_Safe:=TRUE;
Positive_Fit_Safe1:=TRUE;
Positive_Fit_Safe2:=TRUE;
Positive_Fit_Safe3:=TRUE;
Positive_Fit_Safe4:=TRUE;
	step:=370;
END_IF

370:
IF Positive4_Safe THEN
	Positive4_Safe:=FALSE;
	step:=380;
END_IF

380:(*位置4安全--------到工位位置*)
D1:=A1_W1;(*左等待放料工位------下的位置*)
Axis1_MoveAbsolute:=TRUE;
IF Axis1_Abs_Function.Done THEN
Axis1_MoveAbsolute:=FALSE;
Positive3_Safe:=TRUE;
step:=390;
END_IF;

390:(*判断位置1-----------是否安全*)
IF Positive1_Safe THEN
Positive1_Safe:=FALSE;
Y1_6:=FALSE;
step:=400;
END_IF

400:
IF X4_11 THEN
Positive4_Safe:=TRUE;
	step:=10;
END_IF



600:
    IF bstart1   AND NOT Total_Axis_Error  AND NOT total_pausestatus THEN
	step:=bak_step;
END_IF;






(*NG处理流程step*)
2000:(*拍照位置1NG------------处理*)
IF Positive_Camera_Safe2 THEN
Positive_Camera_Safe2:=FALSE;
step:=2010;
END_IF

2010:(*移动到位置2*)
D1:=A1_W3; (*拍照工位2*)
Axis1_MoveAbsolute:=TRUE;
IF Axis1_Abs_Function.Done THEN
Axis1_MoveAbsolute:=FALSE;
(*到位拍照*)
step:=2020;
END_IF

2020:(*拍照位置2------ng处理*)
IF Positive_Camera_Safe3 THEN
Positive_Camera_Safe3:=FALSE;
step:=2040;
END_IF

2040:(*移动到位置2*)
D1:=A1_W4; (*拍照工位3*)
Axis1_MoveAbsolute:=TRUE;
IF Axis1_Abs_Function.Done THEN
Axis1_MoveAbsolute:=FALSE;
(*到位拍照*)
step:=2050;
END_IF

2050:(*拍照位置2------ng处理*)
IF Positive_Camera_Safe4 THEN
Positive_Camera_Safe4:=FALSE;
step:=2060;
END_IF

2060:(*移动到位置2*)
D1:=A1_W5; (*拍照工位3*)
Axis1_MoveAbsolute:=TRUE;
IF Axis1_Abs_Function.Done THEN
Axis1_MoveAbsolute:=FALSE;
Positive1_Safe:=TRUE;
(*到位拍照*)
step:=2070;
END_IF

2070:(*拍照*)
IF Positive_Fit_Safe1 THEN
Positive_Fit_Safe1:=FALSE;
step:=2080;
END_IF

2080:(*到工作位置1*)
D1:=A1_W6;(*工作位置工位1*)
Axis1_MoveAbsolute:=TRUE;
IF Axis1_Abs_Function.Done THEN
Positive_Camera_Safe1:=TRUE;(*工作位置1是给出拍照位置1安全安全位置-------------------------------------*)
Axis1_MoveAbsolute:=FALSE;
step:=2090;
END_IF

2090:(*拍照*)
IF Positive_Fit_Safe2 THEN
Positive_Fit_Safe2:=FALSE;
step:=2100;
END_IF

2100:(*到工作位置1*)
D1:=A1_W7;(*工作位置工位1*)
Axis1_MoveAbsolute:=TRUE;
IF Axis1_Abs_Function.Done THEN
Positive_Camera_Safe2:=TRUE;(*工作位置1是给出拍照位置1安全安全位置-------------------------------------*)
Axis1_MoveAbsolute:=FALSE;
step:=2110;
END_IF

2110:
IF Positive_Fit_Safe3 THEN
Positive_Fit_Safe3:=FALSE;
step:=2120;
END_IF

2120:(*到工作位置1*)
D1:=A1_W8;(*工作位置工位1*)
Axis1_MoveAbsolute:=TRUE;
IF Axis1_Abs_Function.Done THEN
Positive_Camera_Safe3:=TRUE;(*工作位置1是给出拍照位置1安全安全位置-------------------------------------*)
Axis1_MoveAbsolute:=FALSE;
step:=2130;
END_IF

2130:
IF Positive_Fit_Safe4 THEN
Positive_Fit_Safe4:=FALSE;
step:=2140;
END_IF

2140:(*到工作位置1*)
D1:=A1_W9;(*工作位置工位1*)
Axis1_MoveAbsolute:=TRUE;
IF Axis1_Abs_Function.Done THEN
Positive_Camera_Safe4:=TRUE;(*工作位置1是给出拍照位置1安全安全位置-------------------------------------*)
Axis1_MoveAbsolute:=FALSE;
step:=2150;
END_IF

2150:(*贴合位置4状态此时询问位置2是否安全*)
IF Positive2_Safe THEN
	Positive2_Safe:=FALSE;
	step:=350;(*此位置寻味位置3是否安全-------------跳转*)
END_IF










END_CASE


rt_hold(CLK:=( Total_Axis_Error OR  bhold1) , Q=> ); (*暂停状态*)
IF step<>0 AND step<>600   AND  rt_hold.Q THEN
     bak_step:=step;
     step:=600;
END_IF

IF Total_Emergency THEN
Y0_2:=FALSE;
Y0_5:=FALSE;
Left_Translation_Run_1:=FALSE;
Process_2_Can_Push:=FALSE;(*告知上料部分可以上料*)
Can_Move_Film:=FALSE;
Tray1_Have:=FALSE;
Camera_1_1_run:=FALSE;
Camera_1_2_run:=FALSE;
Camera_1_3_run:=FALSE;
Camera_1_4_run:=FALSE;
Camera_1_1_OK:=FALSE;
Camera_1_2_OK:=FALSE;
Camera_1_3_OK:=FALSE;
Camera_1_4_OK:=FALSE;
Positive1_Safe:=FALSE;
Positive2_Safe:=FALSE;
Positive3_Safe:=FALSE;
Positive4_Safe:=FALSE;
Positive_Camera_Safe1:=FALSE;
Positive_Camera_Safe2:=FALSE;
Positive_Camera_Safe3:=FALSE;
Positive_Camera_Safe4:=FALSE;
Positive_Fit_Safe1:=FALSE;
Positive_Fit_Safe2:=FALSE;
Positive_Fit_Safe3:=FALSE;
Positive_Fit_Safe4:=FALSE;
FG_Ready_1:=FALSE;
FG_Ready_2:=FALSE;
FG_Ready_3:=FALSE;
FG_Ready_4:=FALSE;
HB_Fit_Finish_1:=FALSE;
HB_Fit_Finish_2:=FALSE;
HB_Fit_Finish_3:=FALSE;
HB_Fit_Finish_4:=FALSE;
Wait_Robort2_Touch_Finish:=FALSE;
Get_Robot1_Get_Finish:=FALSE;
Process_2_Set_Finish1:=FALSE;(*给机械手可贴合信号*)
Process_2_Can_Push1:=FALSE;
Process_2_Can_Push2:=FALSE;




bak_step:=0;
step:=0;
END_IF
END_PROGRAM

(* POU Run_Main_Folder/Left_Translation/New_Table_2, ST *)
PROGRAM New_Table_2
VAR
	step: INT;
	bak_step:INT;
	rt_hold: R_TRIG;
	UP1: R_TRIG;
	Run_Time:BOOL;
	T1:TON;
	Run_Time_Lreal: TIME;




	T2: TON;
	T3: TON;

END_VAR

VAR_INPUT
	bstart1: BOOL;
	bhold1: BOOL;
	breset1: BOOL;

END_VAR
(*滑台2程序*)


UP1(CLK:=Left_Translation_Run_2 , Q=> );

CASE step OF
0:
 IF UP1.Q THEN
step:=10;
END_IF

10:
D1_1:=A11_W1;(*左等待放料工位*)
Axis11_MoveAbsolute:=TRUE;
IF Axis11_Abs_Function.Done THEN
Axis11_MoveAbsolute:=FALSE;
step:=20;
END_IF;

20:(*到下初始位置------寻味位置1是否安全*)
IF Positive1_Safe THEN
	Positive1_Safe:=FALSE;
	Y1_7:=TRUE;
step:=30;
END_IF

30:
IF X4_13 THEN
	Positive4_Safe:=TRUE;
	step:=40;
END_IF

40:(*安全之后上顶*)
IF Tray2_Have THEN
	step:=72;
ELSE
step:=50;
END_IF

50:(*到位置之后，告知可以放料*)
D1_1:=A11_W1;(*左等待放料工位*)
Axis11_MoveAbsolute:=TRUE;
IF Axis11_Abs_Function.Done THEN
Process_2_Can_Push2:=TRUE;
Axis11_MoveAbsolute:=FALSE;
step:=60;
END_IF;

60:(*上料-----等待放下之后---------*)
IF Process_1_Push_Finish THEN
Tray2_Have:=TRUE;
Process_1_Push_Finish:=FALSE;
step:=70;
END_IF

70:
T2(IN:=TRUE , PT:=t#0.5s , Q=> , ET=> );
   IF T2.Q AND NOT Total_Pause  THEN
T2(IN:=FALSE, PT:=t#0.5S , Q=> , ET=> );
Can_Move_Film:=TRUE;(*给出可撕膜信号*)
step:=71;
END_IF

71:(*撕膜完成信号等到*)
IF Process_1_Push_Finish_Sure THEN
Process_1_Push_Finish_Sure:=FALSE;
step:=72;
END_IF

72:(*判断拍照位置1是否安全*)
IF Positive_Camera_Safe1 THEN
Positive_Camera_Safe1:=FALSE;(*拍照位置1被占据*)
step:=73;
END_IF

73:
D1_1:=A11_W2;(*拍照工位1*)
Axis11_MoveAbsolute:=TRUE;
IF Axis11_Abs_Function.Done THEN
Axis11_MoveAbsolute:=FALSE;
(*到位拍照*)
Camera_1_5_run:=TRUE;
step:=80;
END_IF

80:(*拍照工位1拍照结束-----等待*)
IF Camera_1_5_OK THEN
Camera_1_5_run:=FALSE;
Camera_1_5_OK:=FALSE;
step:=90;
END_IF
IF Camera1_NG THEN  (*拍照失败的处理，判断ng,此时需要给出结果，，，，，，，同时运动到工作位置*)
Camera_1_5_run:=FALSE;
Tray2_Have:=FALSE;
Camera1_NG:=FALSE;
Y0_2:=FALSE;
step:=2000;
END_IF

90:(*判断拍照位置2是否安全*)
IF Positive_Camera_Safe2 THEN
Positive_Camera_Safe2:=FALSE;
step:=100;
END_IF

100:(*移动到位置2*)
D1_1:=A11_W3; (*拍照工位2*)
Axis11_MoveAbsolute:=TRUE;
IF Axis11_Abs_Function.Done THEN
Axis11_MoveAbsolute:=FALSE;
(*到位拍照*)
Camera_1_6_run:=TRUE;
step:=110;
END_IF

110:
IF Camera_1_6_OK THEN
Camera_1_6_run:=FALSE;
Camera_1_6_OK:=FALSE;
step:=120;
END_IF
IF Camera1_NG THEN  (*拍照失败的处理，判断ng,此时需要给出结果，，，，，，，同时运动到工作位置*)
Camera_1_6_run:=FALSE;
Tray2_Have:=FALSE;
Camera1_NG:=FALSE;
Y0_2:=FALSE;
step:=2020;
END_IF


120:(*判断位置3是否安全*)
IF Positive_Camera_Safe3 THEN
Positive_Camera_Safe3:=FALSE;
step:=130;
END_IF

130:(*到工位3*)
D1_1:=A11_W4;(*拍照工位3*)
Axis11_MoveAbsolute:=TRUE;
IF Axis11_Abs_Function.Done THEN
Axis11_MoveAbsolute:=FALSE;
(*到位拍照*)
Camera_1_7_run:=TRUE;
step:=140;
END_IF

140:
IF Camera_1_7_OK THEN
Camera_1_7_run:=FALSE;
Camera_1_7_OK:=FALSE;
step:=150;
END_IF
IF Camera1_NG THEN  (*拍照失败的处理，判断ng,此时需要给出结果，，，，，，，同时运动到工作位置*)
Camera_1_7_run:=FALSE;
Tray2_Have:=FALSE;
Camera1_NG:=FALSE;
Y0_2:=FALSE;
step:=2050;
END_IF

150:(*拍照位置3判断是否安全----------*)
IF Positive_Camera_Safe4 THEN
Positive_Camera_Safe4:=FALSE;
step:=160;
END_IF

160:
D1_1:=A11_W5;(*拍照工位4*)
Axis11_MoveAbsolute:=TRUE;
IF Axis11_Abs_Function.Done THEN
Axis11_MoveAbsolute:=FALSE;
(*到位拍照*)
Camera_1_8_run:=TRUE;

Positive1_Safe:=TRUE;
step:=170;
END_IF

170:
IF Camera_1_8_OK THEN
Camera_1_8_run:=FALSE;
Camera_1_8_OK:=FALSE;
step:=180;
END_IF
IF Camera1_NG THEN  (*拍照失败的处理，判断ng,此时需要给出结果，，，，，，，同时运动到工作位置*)
Camera_1_8_run:=FALSE;
Tray2_Have:=FALSE;
Camera1_NG:=FALSE;
Y0_2:=FALSE;
step:=2070;
END_IF

180:(*判断工作位置1是否安全*)
IF Positive_Fit_Safe1 THEN
Positive_Fit_Safe1:=FALSE;
(*
HB_Fit_Finish_5:=FALSE;
HB_Fit_Finish_6:=FALSE;
HB_Fit_Finish_7:=FALSE;
HB_Fit_Finish_8:=FALSE;*)
step:=190;
END_IF

190:(*到工作位置1*)
D1_1:=A11_W6;(*工作位置工位1*)
Axis11_MoveAbsolute:=TRUE;
IF Axis11_Abs_Function.Done THEN
Axis11_MoveAbsolute:=FALSE;

Positive_Camera_Safe1:=TRUE;(*工作位置1是给出拍照位置1安全安全位置-------------------------------------*)
Process_2_Set_Finish2:=TRUE;(*给机械手可贴合信号*)

FG_Ready_5:=TRUE;
step:=200;
END_IF

200:(*到位等待贴合完成*)
IF HB_Fit_Finish_5 THEN
FG_Ready_5:=FALSE;
HB_Fit_Finish_5:=FALSE;
step:=210;
END_IF

210:(*工位1贴合完成-----询问工作位置2是否安全*)
IF Positive_Fit_Safe2 THEN
Positive_Fit_Safe2:=FALSE;
step:=220;
END_IF

220:(*位置安全------到贴合位置2*)
D1_1:=A11_W7;(*工作位置工位1*)
Axis11_MoveAbsolute:=TRUE;
IF Axis11_Abs_Function.Done THEN
Axis11_MoveAbsolute:=FALSE;

Positive_Camera_Safe2:=TRUE;(*工作位置1是给出拍照位置1安全安全位置-------------------------------------*)

FG_Ready_6:=TRUE;
step:=230;
END_IF

230:(*等待贴合完成信号*)
IF HB_Fit_Finish_6 THEN
FG_Ready_6:=FALSE;
HB_Fit_Finish_6:=FALSE;
step:=240;
END_IF

240:(*贴合完成------寻问位置3是否安全*)
IF Positive_Fit_Safe3 THEN
Positive_Fit_Safe3:=FALSE;
step:=250;
END_IF

250:(*位置安全------到贴合位置2*)
D1_1:=A11_W8;(*工作位置工位1*)
Axis11_MoveAbsolute:=TRUE;
IF Axis11_Abs_Function.Done THEN
Axis11_MoveAbsolute:=FALSE;

Positive_Camera_Safe3:=TRUE;(*工作位置1是给出拍照位置1安全安全位置-------------------------------------*)

FG_Ready_7:=TRUE;
step:=260;
END_IF

260:(*等待贴合完成信号*)
IF HB_Fit_Finish_7 THEN
FG_Ready_7:=FALSE;
HB_Fit_Finish_7:=FALSE;
step:=270;
END_IF

270:(*位置3贴合完成，询问位置4是否安全*)
IF Positive_Fit_Safe4 THEN
Positive_Fit_Safe4:=FALSE;
step:=280;
END_IF

280:(*位置安全------到贴合位置2*)
D1_1:=A11_W9;(*工作位置工位1*)
Axis11_MoveAbsolute:=TRUE;
IF Axis11_Abs_Function.Done THEN
Axis11_MoveAbsolute:=FALSE;

Positive_Camera_Safe4:=TRUE;(*工作位置1是给出拍照位置1安全安全位置-------------------------------------*)
Process_2_Set_Finish2:=FALSE;(*给机械手可贴合信号*)

FG_Ready_8:=TRUE;
step:=290;
END_IF

290:(*等待贴合完成信号*)
IF HB_Fit_Finish_8 THEN
FG_Ready_8:=FALSE;
HB_Fit_Finish_8:=FALSE;
step:=300;
END_IF

300:
IF Positive2_Safe THEN
	Positive2_Safe:=FALSE;
	step:=310;
END_IF

310:(*位置到位后，等待，送吸嘴*)
IF Wait_Robort2_Touch_Finish  THEN
Wait_Robort2_Touch_Finish:=FALSE;
Y0_2:=FALSE;
step:=320;
END_IF

320:
T3(IN:=TRUE , PT:=t#1s , Q=> , ET=> );
   IF T3.Q AND NOT Total_Pause  THEN
T3(IN:=FALSE, PT:=t#1S , Q=> , ET=> );
step:=340;
END_IF

340:
IF Get_Robot1_Get_Finish THEN
Tray2_Have:=FALSE;
Get_Robot1_Get_Finish:=FALSE;
step:=350;
END_IF

350:
IF Positive3_Safe THEN
	Positive3_Safe:=FALSE;
	Y1_7:=FALSE;
	step:=360;
END_IF

360:
IF X4_14 THEN
Positive2_Safe:=TRUE;
Positive_Fit_Safe1:=TRUE;
Positive_Fit_Safe2:=TRUE;
Positive_Fit_Safe3:=TRUE;
Positive_Fit_Safe4:=TRUE;

	step:=370;
END_IF

370:(*下降之后，*)
IF Positive4_Safe THEN
	Positive4_Safe:=FALSE;
	step:=380;
END_IF

380:
D1_1:=A11_W1;(*左等待放料工位------下的位置*)
Axis11_MoveAbsolute:=TRUE;
IF Axis11_Abs_Function.Done THEN
Axis11_MoveAbsolute:=FALSE;
Positive3_Safe:=TRUE;
step:=10;
END_IF;



600:
    IF bstart1   AND NOT Total_Axis_Error  AND NOT total_pausestatus  THEN
	step:=bak_step;
END_IF;







2000:(*拍照位置1NG------------处理*)
IF Positive_Camera_Safe2 THEN
Positive_Camera_Safe2:=FALSE;
step:=2010;
END_IF

2010:(*移动到位置2*)
D1_1:=A11_W3; (*拍照工位2*)
Axis11_MoveAbsolute:=TRUE;
IF Axis11_Abs_Function.Done THEN
Axis11_MoveAbsolute:=FALSE;
(*到位拍照*)
step:=2020;
END_IF

2020:(*拍照位置2------ng处理*)
IF Positive_Camera_Safe3 THEN
Positive_Camera_Safe3:=FALSE;
step:=2040;
END_IF

2040:(*移动到位置2*)
D1_1:=A11_W4; (*拍照工位3*)
Axis11_MoveAbsolute:=TRUE;
IF Axis11_Abs_Function.Done THEN
Axis11_MoveAbsolute:=FALSE;
(*到位拍照*)
step:=2050;
END_IF

2050:(*拍照位置2------ng处理*)
IF Positive_Camera_Safe4 THEN
Positive_Camera_Safe4:=FALSE;
step:=2060;
END_IF

2060:(*移动到位置2*)
D1_1:=A11_W5; (*拍照工位3*)
Axis11_MoveAbsolute:=TRUE;
IF Axis11_Abs_Function.Done THEN
Axis11_MoveAbsolute:=FALSE;
Positive1_Safe:=TRUE;
(*到位拍照*)
step:=2070;
END_IF

2070:(*拍照*)
IF Positive_Fit_Safe1 THEN
Positive_Fit_Safe1:=FALSE;
step:=2080;
END_IF

2080:(*到工作位置1*)
D1_1:=A11_W6;(*工作位置工位1*)
Axis11_MoveAbsolute:=TRUE;
IF Axis11_Abs_Function.Done THEN
Positive_Camera_Safe1:=TRUE;(*工作位置1是给出拍照位置1安全安全位置-------------------------------------*)
Axis11_MoveAbsolute:=FALSE;
step:=2090;
END_IF

2090:(*拍照*)
IF Positive_Fit_Safe2 THEN
Positive_Fit_Safe2:=FALSE;
step:=2100;
END_IF

2100:(*到工作位置1*)
D1_1:=A11_W7;(*工作位置工位1*)
Axis11_MoveAbsolute:=TRUE;
IF Axis11_Abs_Function.Done THEN
Positive_Camera_Safe2:=TRUE;(*工作位置1是给出拍照位置1安全安全位置-------------------------------------*)
Axis11_MoveAbsolute:=FALSE;
step:=2110;
END_IF

2110:
IF Positive_Fit_Safe3 THEN
Positive_Fit_Safe3:=FALSE;
step:=2120;
END_IF

2120:(*到工作位置1*)
D1_1:=A11_W8;(*工作位置工位1*)
Axis11_MoveAbsolute:=TRUE;
IF Axis11_Abs_Function.Done THEN
Positive_Camera_Safe3:=TRUE;(*工作位置1是给出拍照位置1安全安全位置-------------------------------------*)
Axis11_MoveAbsolute:=FALSE;
step:=2130;
END_IF

2130:
IF Positive_Fit_Safe4 THEN
Positive_Fit_Safe4:=FALSE;
step:=2140;
END_IF

2140:(*到工作位置1*)
D1_1:=A11_W9;(*工作位置工位1*)
Axis11_MoveAbsolute:=TRUE;
IF Axis11_Abs_Function.Done THEN
Positive_Camera_Safe4:=TRUE;(*工作位置1是给出拍照位置1安全安全位置-------------------------------------*)
Axis11_MoveAbsolute:=FALSE;
step:=2150;
END_IF

2150:(*贴合位置4状态此时询问位置2是否安全*)
IF Positive2_Safe THEN
	Positive2_Safe:=FALSE;
	step:=350;(*此位置寻味位置3是否安全-------------跳转*)
END_IF



END_CASE



rt_hold(CLK:=( Total_Axis_Error OR  bhold1) , Q=> ); (*暂停状态*)
IF step<>0 AND step<>600   AND  rt_hold.Q THEN
     bak_step:=step;
     step:=600;
END_IF

IF Total_Emergency THEN
Left_Translation_Run_2:=FALSE;
Process_2_Can_Push:=FALSE;(*告知上料部分可以上料*)
Can_Move_Film:=FALSE;
Tray2_Have:=FALSE;

Camera_1_5_run:=FALSE;
Camera_1_6_run:=FALSE;
Camera_1_7_run:=FALSE;
Camera_1_8_run:=FALSE;
Positive1_Safe:=FALSE;
Positive2_Safe:=FALSE;
Positive3_Safe:=FALSE;
Positive4_Safe:=FALSE;
Camera_1_5_OK:=FALSE;
Camera_1_6_OK:=FALSE;
Camera_1_7_OK:=FALSE;
Camera_1_8_OK:=FALSE;

Positive_Fit_Safe1:=FALSE;
Positive_Fit_Safe2:=FALSE;
Positive_Fit_Safe3:=FALSE;
Positive_Fit_Safe4:=FALSE;
FG_Ready_5:=FALSE;
FG_Ready_6:=FALSE;
FG_Ready_7:=FALSE;
FG_Ready_8:=FALSE;
HB_Fit_Finish_5:=FALSE;
HB_Fit_Finish_6:=FALSE;
HB_Fit_Finish_7:=FALSE;
HB_Fit_Finish_8:=FALSE;
Wait_Robort2_Touch_Finish:=FALSE;
Get_Robot1_Get_Finish:=FALSE;
Process_2_Set_Finish2:=FALSE;(*给机械手可贴合信号*)



bak_step:=0;
step:=0;
END_IF
END_PROGRAM

(* POU Test_Part_pro/Film_Test1, ST *)
PROGRAM Film_Test1
VAR
	UP1: R_TRIG;
	UP2: R_TRIG;
	T1:TON;

	step:INT;



	T2: TON;
	T3: TON;
	T4: TON;
	T5:TON;

	T104: TON;
END_VAR
UP1(CLK:=Film_Test , Q=> );


CASE step OF
0:
 IF UP1.Q  THEN
step:=7;
END_IF

7:
IF Film_Once_Run THEN
Film_Once_Run:=FALSE;
step:=10;
END_IF



10:(*到放料工位置，取料*)
Y0_5:=FALSE;
D4:=A4_W4;(*到放料工位，等到是否可以放料，*)
Axis4_MoveAbsolute:=TRUE;
IF Axis4_Abs_Function.Done THEN
Axis4_MoveAbsolute:=FALSE;
step:=20;
END_IF

20:(*放料工位，下降工位*)
D5:=A5_W4;
Axis5_MoveAbsolute:=TRUE;
IF Axis5_Abs_Function.Done THEN
Axis5_MoveAbsolute:=FALSE;
Y0_3:=TRUE;
step:=30;
END_IF

30:(*吸取，料，上抬，*)
T2(IN:=TRUE , PT:=t#1s , Q=> , ET=> );
   IF T2.Q AND NOT Total_Pause  THEN
T2(IN:=FALSE, PT:=t#1S , Q=> , ET=> );
step:=40;
END_IF

40:(*吸取之后，上抬*)
D5:=A5_W0;
Axis5_MoveAbsolute:=TRUE;
IF Axis5_Abs_Function.Done THEN
Axis5_MoveAbsolute:=FALSE;
Y0_5:=TRUE;
Y0_4:=TRUE;
step:=50;
END_IF

50:(*吸取之后，气缸做动作*)
T3(IN:=TRUE , PT:=t#1s , Q=> , ET=> );
   IF T3.Q AND NOT Total_Pause  THEN
T3(IN:=FALSE, PT:=t#1S , Q=> , ET=> );
Y1_4:=TRUE;
step:=60;
END_IF

60:
T4(IN:=TRUE , PT:=t#1s , Q=> , ET=> );
   IF T4.Q AND NOT Total_Pause  THEN
T4(IN:=FALSE, PT:=t#1S , Q=> , ET=> );
step:=70;
END_IF


70:(*上料可以之后，到放料下降工位*)
D5:=A5_W4;
Axis5_MoveAbsolute:=TRUE;
IF Axis5_Abs_Function.Done THEN
Axis5_MoveAbsolute:=FALSE;
Y0_3:=FALSE;
step:=110;
END_IF

110:
T5(IN:=TRUE , PT:=t#0.2s , Q=> , ET=> );
   IF T5.Q AND NOT Total_Pause  THEN
T5(IN:=FALSE, PT:=t#0.2S , Q=> , ET=> );
step:=120;
END_IF

120:
IF Qurensimo THEN(*接收到撕膜信号之后，正式开始撕膜*)
Qurensimo:=FALSE;
step:=130;
END_IF

130:
D15_1:=10;
D5:=A5_W5;(*撕膜Z轴上抬一点---------*)
Axis5_1_MoveAbsolute:=TRUE;
IF Axis5_1_Abs_Function.Done THEN
Axis5_1_MoveAbsolute:=FALSE;
step:=140;
END_IF

140:(*联动*)
D14_1:=40;
D15_1:=5;
D4:=A4_W5;
D5:=A5_W6;
Axis4_1_MoveAbsolute:=TRUE;
Axis5_1_MoveAbsolute:=TRUE;
IF Axis4_1_Abs_Function.Done  AND Axis5_1_Abs_Function.Done THEN
Axis4_1_MoveAbsolute:=FALSE;
Axis5_1_MoveAbsolute:=FALSE;
step:=150;
END_IF

150:(*联动结束-------------集训动作保证进入非料盘位置*)
D15_1:=70;
D5:=A5_W8;(*Z轴上抬点位*)
Axis5_1_MoveAbsolute:=TRUE;
IF  Axis5_1_Abs_Function.Done THEN
Axis5_1_MoveAbsolute:=FALSE;
step:=160;
END_IF

160:(*丢么位置坐标*)
D4:=A4_W3;
Axis4_MoveAbsolute:=TRUE;
IF Axis4_Abs_Function.Done THEN
Axis4_MoveAbsolute:=FALSE;
step:=170;
END_IF

170:(*丢么下降位置*)
D5:=A5_W3;
Axis5_MoveAbsolute:=TRUE;
IF   Axis5_Abs_Function.Done THEN
Axis5_MoveAbsolute:=FALSE;
Y1_4:=FALSE;(*JIAZI*)
Y0_4:=FALSE;
step:=180;
END_IF

180:
T104(IN:=TRUE , PT:=t#0.8s , Q=> , ET=> );
   IF T104.Q AND NOT Total_Pause  THEN
T104(IN:=FALSE, PT:=t#0.8S , Q=> , ET=> );
step:=190;
END_IF

190:(*丢么位置丢弃费膜，结束，到吸取料位置*)
D5:=A5_W0;
Axis5_MoveAbsolute:=TRUE;
IF Axis5_Abs_Function.Done THEN
Axis5_MoveAbsolute:=FALSE;
step:=200;
END_IF

200:
D4:=A4_W1;(*取料位置等待*)
Axis4_MoveAbsolute:=TRUE;
IF Axis4_Abs_Function.Done THEN
Axis4_MoveAbsolute:=FALSE;
step:=7;
END_IF


END_CASE


IF Film_Test_OFF THEN
Film_Test:=FALSE;
step:=0;

END_IF
END_PROGRAM

(* POU Test_Part_pro/Rool_Test, ST *)
PROGRAM Rool_Test
VAR
	step: INT;
	bak_step:INT;
	rt_hold: R_TRIG;
	UP1: R_TRIG;
	T1: TON;
	T2:TON;

	Rool_Test_Run: BOOL;
	Button_Test: BOOL;
END_VAR
UP1(CLK:=Rool_Test_Run , Q=> );

CASE step OF
0:
 IF UP1.Q THEN
step:=10;
END_IF

10:(*滚压部分开始动作*)
(*判断机械手是否放好料---------放好之后，进行滚压动作，询问右移载是否可以送料，可送料之后，给出料，同时，发出，给料完成信号*)
IF Button_Test THEN
Button_Test:=FALSE;

	step:=20;
END_IF

20:(*无料的操作*)
D10:=A10_W2;
Axis10_MoveAbsolute:=TRUE;
IF Axis10_Abs_Function.Done THEN
Axis10_MoveAbsolute:=FALSE;
step:=40;
END_IF


40:(*准备推入气缸*)
T1(IN:=TRUE , PT:=t#0.1s , Q=> , ET=> );
   IF T1.Q   THEN
T1(IN:=FALSE, PT:=t#0.1S , Q=> , ET=> );
Y0_10:=TRUE;(*推入气缸*)
step:=50;
END_IF

50:
IF X2_16 THEN
Y0_9:=TRUE;
Y0_11:=TRUE;
step:=60;
END_IF

60:
IF X3_2  THEN(*压合气缸到位，等待滚压*)
Rolling_Number:=0;
step:=70;
END_IF

70:
D10:=A10_W1;(*出去位置*)
Axis10_MoveAbsolute:=TRUE;
IF Axis10_Abs_Function.Done THEN
Axis10_MoveAbsolute:=FALSE;
step:=80;
END_IF

80:
D10:=A10_W2;
Axis10_MoveAbsolute:=TRUE;
IF Axis10_Abs_Function.Done THEN
Axis10_MoveAbsolute:=FALSE;
Rolling_Number:=Rolling_Number+1;
step:=90;
END_IF

90:
IF Rolling_Number>=Set_Rolling_Number THEN
Rolling_Number:=0;
Y0_11:=FALSE;
Y0_9:=FALSE;
step:=100;(*次数满足，跳转*)
ELSE
step:=70;
END_IF

100:
IF X3_3 THEN
Y0_10:=FALSE;
step:=110;
END_IF

110:
IF X3_1 THEN
step:=10;
END_IF

END_CASE
END_PROGRAM

(* POU Run_Main_Folder/Right_Tray_Pro/Liftin_Feed_Right_Down, ST *)
PROGRAM Liftin_Feed_Right_Down
VAR

	step: INT;
	bak_step:INT;
	rt_hold: R_TRIG;
	UP1: R_TRIG;
	T1: TON;
	T2:TON;
	DOWN1: F_TRIG;
	lastHeight:LREAL;

END_VAR

VAR_INPUT
	bstart1: BOOL;
	bhold1: BOOL;
	breset1: BOOL;

END_VAR
(*完成品下料程序*)

UP1(CLK:=Liftin_Feed_Right_1_Run , Q=> );(**)

CASE step OF
0:
 IF UP1.Q THEN
step:=10;
END_IF


10:(*上升运行*)
Axis8_PTF_2:=TRUE;
IF X2_4 AND  X1_3 THEN(*碰到光纤，同时没有碰到极限，此时上料ok*)
Axis8_PTF_2:=FALSE;
Axis8_Halt:=TRUE;
lastHeight:=axis8.NcToPlc.ActPos;
step:=30;
END_IF
IF NOT X1_3 THEN(*碰到极限，此时表示料空*)
Axis8_PTF_2:=FALSE;
Axis8_Halt:=TRUE;
step:=120;
END_IF



20:(*碰到本来就有料的情况，，，，此时等待放满信号*)
Axis8_Halt:=FALSE;
IF Get_Robort3_Tray_Full THEN

Feed_3_Finish:=FALSE;
Get_Robort3_Tray_Full:=FALSE;
lastHeight:=axis8.NcToPlc.ActPos;
step:=30;
END_IF

30:(*准备下降*)
Axis8_Halt:=FALSE;
(*接收到可降信号，开始下降，到传感器下降沿停止下降，等待*)
IF x2_4  THEN
	step:=31;
ELSE
	step:=32;
END_IF

31:
	Axis8_PTF:=TRUE;
	DOWN1(CLK:=X2_4 , Q=> );
	IF DOWN1.Q  AND NOT  (axis8.NcToPlc.ActPos<=50) THEN
	Axis8_PTF:=FALSE;
	Right_Need_Tray:=TRUE;
	Axis8_Halt:=TRUE;
	step:=40;
	END_IF
	IF  (axis8.NcToPlc.ActPos<=50) THEN(*碰到极限，此时表示料空------此时表示需要上料*)
	Axis8_PTF:=FALSE;
	Axis8_Halt:=TRUE;
	step:=400;
	END_IF

32:
	Axis8_PTF:=TRUE;

	IF  ((lastHeight-axis8.NcToPlc.ActPos)>=3) AND NOT  (axis8.NcToPlc.ActPos<=50) THEN
	Axis8_PTF:=FALSE;
	Right_Need_Tray:=TRUE;
	Axis8_Halt:=TRUE;
	step:=40;
	END_IF
	IF  (axis8.NcToPlc.ActPos<=50) THEN(*碰到极限，此时表示料空------此时表示需要上料*)
	Axis8_PTF:=FALSE;
	Axis8_Halt:=TRUE;
	step:=400;
	END_IF




40:(*电机下降到下降沿以下的时候，给出缺空盘信号，当放料盘ok之后，*)
Axis8_Halt:=FALSE;
IF Right_Send_Tray_OK THEN
Right_Send_Tray_OK:=FALSE;
step:=20;
END_IF

400:(*碰到原点，此时，回到下初始位置，给出料满提示*)
Axis8_Halt:=FALSE;
D8:=D800;
Axis8_MoveAbsolute:=TRUE;
IF Axis8_Abs_Function.Done THEN
Axis8_MoveAbsolute:=FALSE;
Feed_Right_Full_Alam:=TRUE;(*不暂停，只提示*)
step:=50;
END_IF

50:
Axis8_Halt:=FALSE;
IF Right_Down_Button AND NOT Total_Pause THEN
	Right_Down_Button:=FALSE;
Feed_Right_Full_Alam:=FALSE;
	step:=10;(*确认拿走料之后，运动到初始位置*)
END_IF



120:
Axis8_Halt:=FALSE;
D8:=D810;
Axis8_MoveAbsolute:=TRUE;
IF Axis8_Abs_Function.Done THEN
Axis8_MoveAbsolute:=FALSE;
Right_Need_Tray:=TRUE;(*需要移载气缸给出料*)
step:=40;
END_IF

300:
    IF bstart1   AND NOT Total_Axis_Error AND NOT total_pausestatus  THEN
	step:=bak_step;
END_IF;
END_CASE


rt_hold(CLK:=( Total_Axis_Error OR  bhold1) , Q=> ); (*暂停状态*)
IF step<>0 AND step<>300   AND  rt_hold.Q THEN
     bak_step:=step;
     step:=300;
END_IF


IF Right_Down_Button THEN
Right_Down_Button:=FALSE;
END_IF

IF Total_Emergency THEN
Liftin_Feed_Right_1_Run:=FALSE;
Feed_Right_Full_Alam:=FALSE;
Right_Need_Tray:=FALSE;

bak_step:=0;
step:=0;
END_IF


(*随时可以不做料的操作*)
IF Feed_Right_Button1 AND (step=20 OR step=40)  AND NOT Total_Pause THEN
Feed_Right_Button1:=FALSE;
Feed_3_Finish:=FALSE;
Right_Need_Tray:=FALSE;
Get_Robort3_Tray_Full:=FALSE;
step:=400;
ELSE
Feed_Right_Button1:=FALSE;
END_IF
END_PROGRAM

(* POU Run_Main_Folder/Right_Tray_Pro/Liftin_Feed_Right_Up, ST *)
PROGRAM Liftin_Feed_Right_Up
VAR

	step: INT;
	bak_step:INT;
	rt_hold: R_TRIG;
	UP1: R_TRIG;
	DOWN1: F_TRIG;

	T1: TON;
	T2:TON;

END_VAR

VAR_INPUT
	bstart1: BOOL;
	bhold1: BOOL;
	breset1: BOOL;

END_VAR
(*成品空盘供料上料*)

(*左下降，初始化，回原点到初始位置，，，启动之后，先往上走，到初始位置(第一次回原点使用)  ，接收到送料完成可下降信号，则
开始下降，等现将结束，告知，可放料*)

UP1(CLK:=Liftin_Feed_Right_2_Run , Q=> );

CASE step OF
0:
 IF UP1.Q THEN
step:=1;
END_IF

1:
(*初始化之后位置在下面的初始位置*)
Axis9_PTF_2:=TRUE;
IF X2_5 AND X1_6 THEN
Axis9_PTF_2:=FALSE;
Right_Loading_OK:=TRUE;(*碰到光纤，表示到达上料位置，准备好上空料盘*)
Axis9_Halt:=TRUE;
step:=20;
END_IF
IF NOT X1_6 THEN
Axis9_PTF_2:=FALSE;
Axis9_Halt:=TRUE;
step:=50;(*撞到极限，此时需要回到上面的初始位置*)
END_IF


20:(*等到取料完成信号，当完成之后，电机上升，*)
Axis9_Halt:=FALSE;
IF Right_Get_Tray_OK THEN
Right_Get_Tray_OK:=FALSE;
step:=1;
END_IF


50:(*碰到极限，此时需要下降到初始位置*)
Axis9_Halt:=FALSE;
D9:=D900;
Axis9_MoveAbsolute:=TRUE;
IF Axis9_Abs_Function.Done THEN
Axis9_MoveAbsolute:=FALSE;
Feed_Right_None_Alam:=TRUE;(*不暂停，只提示*)
step:=60;
END_IF

60:
Axis9_Halt:=FALSE;
IF Right_Up_Button AND NOT Total_Pause THEN
	Right_Up_Button:=FALSE;
	Feed_Right_None_Alam:=FALSE;
	step:=1;(*确认拿走料之后，运动到初始位置*)
END_IF

300:
    IF bstart1   AND NOT Total_Axis_Error AND NOT total_pausestatus  THEN
	step:=bak_step;
END_IF;
END_CASE


rt_hold(CLK:=( Total_Axis_Error OR  bhold1) , Q=> ); (*暂停状态*)
IF step<>0 AND step<>300   AND  rt_hold.Q THEN
     bak_step:=step;
     step:=300;
END_IF


IF Right_Up_Button THEN
Right_Up_Button:=FALSE;
END_IF

IF Total_Emergency THEN
Liftin_Feed_Right_2_Run:=FALSE;
Right_Loading_OK:=FALSE;
Feed_Right_None_Alam:=FALSE;
Right_Get_Tray_OK:=FALSE;
bak_step:=0;
step:=0;
END_IF


(*随时可以不做料的操作*)
IF Feed_Right_Button2 AND step=20 AND NOT Total_Pause THEN
Feed_Right_Button2:=FALSE;
Right_Loading_OK:=FALSE;

step:=50;
ELSE
Feed_Right_Button2:=FALSE;
END_IF
END_PROGRAM

(* POU Run_Main_Folder/Right_Tray_Pro/Right_Carry_1, ST *)
PROGRAM Right_Carry_1
VAR
	step: INT;
	bak_step:INT;
	rt_hold: R_TRIG;
	UP1: R_TRIG;
	T1: TON;
	TT1: TON;

	T2: TON;

	T8: TON;
END_VAR

VAR_INPUT
	bstart1: BOOL;
	bhold1: BOOL;
	breset1: BOOL;

END_VAR
(*tray盘移载*)

UP1(CLK:=Right_Carry_Run , Q=> );

CASE step OF
0:
 IF UP1.Q THEN
step:=10;
END_IF

(*等待机械手取完信号，当移载完成之后，给左可上升信号，放下料之后给出，左可下降信号*)
10:
IF Right_hand_have THEN (*判断收上是否空料盘*)
(*手上有料，则直接放料位置*)
step:=70;
ELSE
step:=20;
END_IF

20:(*判断是否上料OK--------可取信号*)
IF Right_Loading_OK THEN
Right_Loading_OK:=FALSE;
step:=25;
END_IF


25:(*吸取成功后，判断是否要料*)
IF Right_Need_Tray THEN
Right_Need_Tray:=FALSE;
step:=30;
END_IF

30:
IF NOT  Pressure_Right_Fail THEN
Y1_1:=TRUE;(*上下气缸动作*)
END_IF
IF X3_10 THEN
Y1_2:=TRUE;
step:=50;
END_IF

50:
T1(IN:=TRUE , PT:=t#0.8s , Q=> , ET=> );
   IF T1.Q AND NOT Total_Pause  THEN
T1(IN:=FALSE, PT:=t#0.8S , Q=> , ET=> );
Y1_1:=FALSE;
step:=60;
END_IF

60:
IF X3_11 THEN(*气缸上抬到位*)
step:=68;
END_IF

68:
T8(IN:=TRUE , PT:=t#1s , Q=> , ET=> );
   IF T8.Q AND NOT Total_Pause  THEN
T8(IN:=FALSE, PT:=t#1S , Q=> , ET=> );
step:=70;
END_IF

70:(*判断是否吸取成功*)
IF X3_12 THEN
Right_Get_Tray_OK:=TRUE;
Right_hand_have:=TRUE;
Y0_16:=TRUE;
step:=80;
(*吸取成功*)
ELSE

Pressure_Right_Fail:=TRUE;
step:=30;(*重复吸取-----等待成功*)

END_IF



80:(*成功之后----给出可以上顶*)
IF X3_8 THEN
Y1_1:=TRUE;
step:=90;
END_IF

90:
IF X3_10 THEN
Y1_2:=FALSE;;
step:=95;
END_IF

95:(*放料之后,*)
TT1(IN:=TRUE , PT:=t#0.8s , Q=> , ET=> );
   IF TT1.Q AND NOT Total_Pause  THEN
TT1(IN:=FALSE, PT:=t#0.8S , Q=> , ET=> );
Y1_1:=FALSE;
step:=96;
END_IF

96:
IF X3_11 THEN
Right_hand_have:=FALSE;
Right_Send_Tray_OK:=TRUE;
Y0_16:=FALSE;
step:=97;
END_IF

97:(*恢复之后，给出机械手信号*)
IF X3_9 THEN
Feed_3_Finish:=TRUE;
step:=20;
END_IF



300:
    IF bstart1   AND NOT Total_Axis_Error AND NOT total_pausestatus  THEN
	step:=bak_step;
END_IF;
END_CASE

rt_hold(CLK:=( Total_Axis_Error OR  bhold1) , Q=> ); (*暂停状态*)
IF step<>0 AND step<>300   AND  rt_hold.Q THEN
     bak_step:=step;
     step:=300;
END_IF

IF Total_Emergency THEN
Y1_2:=FALSE;
Right_hand_have:=FALSE;
Right_Carry_Run:=FALSE;
Right_Get_Tray_OK:=FALSE;
Feed_3_Finish:=FALSE;
Right_Loading_OK:=FALSE;
Right_Need_Tray:=FALSE;
bak_step:=0;
step:=0;
END_IF
END_PROGRAM

(* POU PLC_Action/PID2, FBD *)
PROGRAM PID2
VAR
END_VAR
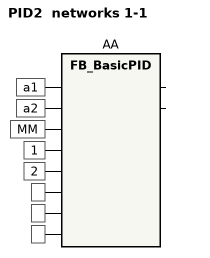
_FBD_ (* Function Block Diagram *)
NETWORK 1
	AA:FB_BasicPID(a1, a2, MM, 1, 2, , , )
_END_FBD_
END_PROGRAM

(* POU PLC_Action/PID1, LD *)
PROGRAM PID1
VAR
END_VAR
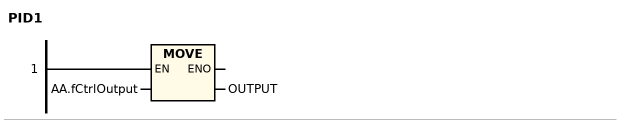
_LD_ (* Ladder Diagram *)
NETWORK 1
	*
		EN --- MOVE(AA.fCtrlOutput) => OUTPUT
_END_LD_
(* the same logic as Structured Text *)
(* Network 1 *)
OUTPUT := AA.fCtrlOutput;
END_PROGRAM

(* POU Debug_Folder/Axis12_Debug_Model, ST *)
PROGRAM Axis12_Debug_Model
VAR

	UP1: R_TRIG;
	UP2: R_TRIG;
	UP3: R_TRIG;
	UP4: R_TRIG;
	step:INT;
END_VAR
UP1(CLK:=Axis12_debug_trigger , Q=> );

CASE step OF
0:
IF UP1.Q THEN
step:=1;
END_IF;

1:
UP2(CLK:=Axis12_mov_add , Q=> );
UP3(CLK:=Axis12_mov_sub , Q=> );
UP4(CLK:=Axis12_mov_line , Q=> );

IF UP2.Q AND Debug_Model AND Axis12_Poweron  AND NOT Total_Pause THEN
D1_2:=Axis12.NcToPlc.ActPos+D200;
Axis12_mov_add:=FALSE;
step:=10;
ELSE
Axis12_mov_add:=FALSE;
Axis12_MoveAbsolute:=FALSE;
END_IF

IF UP3.Q AND Debug_Model AND Axis12_Poweron AND NOT Total_Pause THEN
D1_2:=Axis12.NcToPlc.ActPos-D200;
Axis12_mov_sub:=FALSE;
step:=10;
ELSE
Axis12_mov_sub:=FALSE;
Axis12_MoveAbsolute:=FALSE;
END_IF

IF UP4.Q AND Debug_Model AND Axis12_Poweron  AND NOT Total_Pause THEN
D1_2:=D212;
Axis12_mov_line:=FALSE;
step:=10;
ELSE
Axis12_mov_line:=FALSE;
Axis12_MoveAbsolute:=FALSE;
END_IF

10:
Axis12_MoveAbsolute:=TRUE;
IF Axis12_Abs_Function.Done THEN
Axis12_MoveAbsolute:=FALSE;
step:=1;
END_IF
END_CASE

IF Axis12_mov_add THEN
Axis12_mov_add:=FALSE;
END_IF
IF Axis12_mov_sub THEN
Axis12_mov_sub:=FALSE;
END_IF
IF Axis12_mov_line THEN
Axis12_mov_line:=FALSE;
END_IF


IF NOT Debug_Model  THEN
Axis12_debug_trigger:=FALSE;
step:=0;
END_IF

IF Total_Emergency THEN
Axis12_debug_trigger:=FALSE;
Axis12_mov_add:=FALSE;
Axis12_mov_sub:=FALSE;
Axis12_mov_line:=FALSE;
Axis12_MoveAbsolute:=FALSE;
step:=0;
END_IF
END_PROGRAM

(* POU Other_Folder/Home_Back/Axis12_Home_Back, LD *)
PROGRAM Axis12_Home_Back
VAR
	UP1: R_TRIG;
	M1: BOOL;
	M2: BOOL;
	UP2: R_TRIG;
	T1: TON;
	M3: BOOL;
	M4: BOOL;
	DOWN1: F_TRIG;
	M20: BOOL;
END_VAR
VAR (* helpers for the ST form of the networks *)
	_p1 : BOOL;
	_p2 : BOOL;
	_p3 : BOOL;
END_VAR
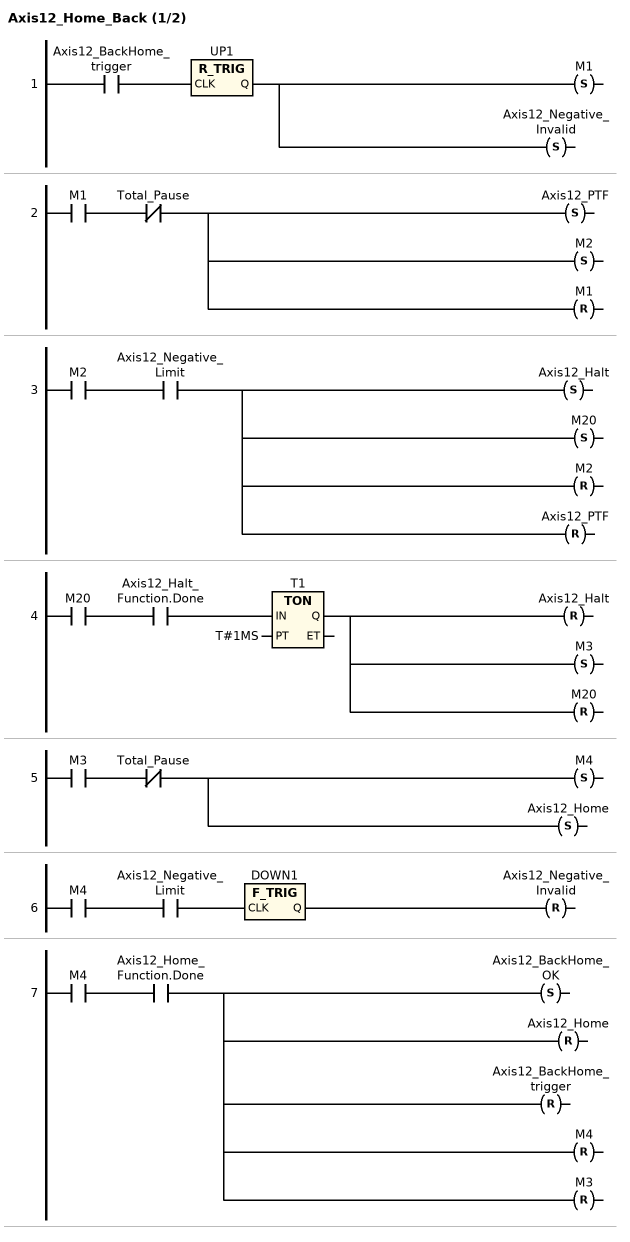
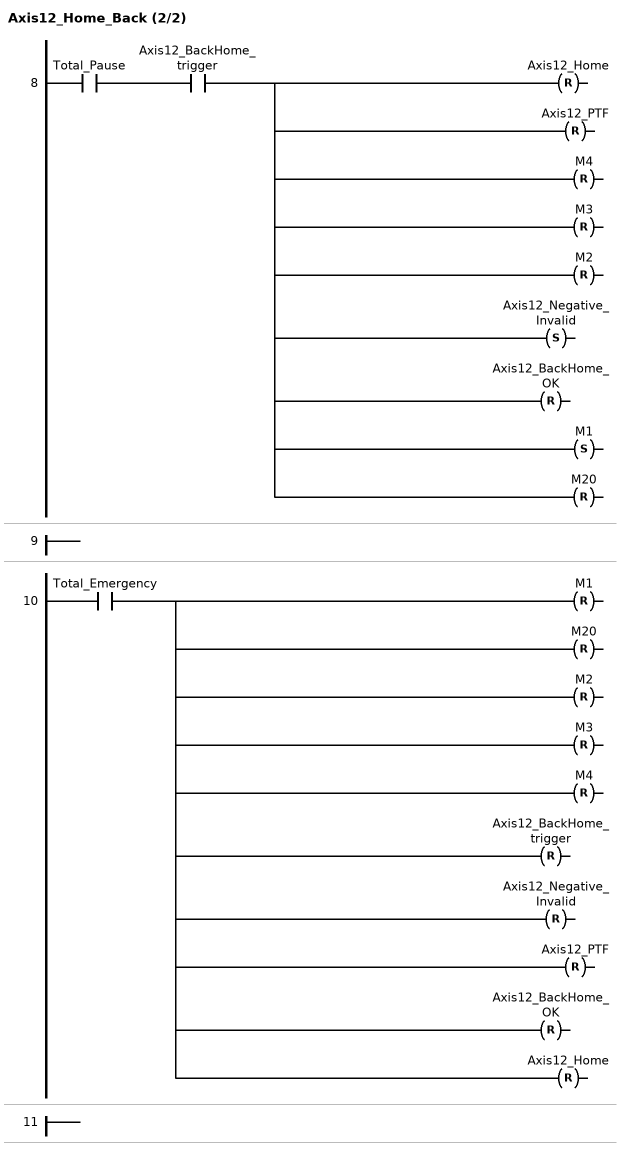
_LD_ (* Ladder Diagram *)
NETWORK 1
	[Axis12_BackHome_trigger] - UP1:R_TRIG(CLK: *) --- (S M1) (S Axis12_Negative_Invalid)
NETWORK 2
	[M1] - [/Total_Pause] --- (S Axis12_PTF) (S M2) (R M1)
NETWORK 3
	[M2] - [Axis12_Negative_Limit] --- (S Axis12_Halt) (S M20) (R M2) (R Axis12_PTF)
NETWORK 4
	[M20] - [Axis12_Halt_Function.Done] - T1:TON(IN: *, PT: T#1MS) --- (R Axis12_Halt) (S M3) (R M20)
NETWORK 5
	[M3] - [/Total_Pause] --- (S M4) (S Axis12_Home)
NETWORK 6
	[M4] - [Axis12_Negative_Limit] - DOWN1:F_TRIG(CLK: *) --- (R Axis12_Negative_Invalid)
NETWORK 7
	[M4] - [Axis12_Home_Function.Done] --- (S Axis12_BackHome_OK) (R Axis12_Home) (R Axis12_BackHome_trigger) (R M4) (R M3)
NETWORK 8
	[Total_Pause] - [Axis12_BackHome_trigger] --- (R Axis12_Home) (R Axis12_PTF) (R M4) (R M3) (R M2) (S Axis12_Negative_Invalid) (R Axis12_BackHome_OK) (S M1) (R M20)
NETWORK 9
	*
NETWORK 10
	[Total_Emergency] --- (R M1) (R M20) (R M2) (R M3) (R M4) (R Axis12_BackHome_trigger) (R Axis12_Negative_Invalid) (R Axis12_PTF) (R Axis12_BackHome_OK) (R Axis12_Home)
NETWORK 11
	*
_END_LD_
(* the same logic as Structured Text *)
(* Network 1 *)
UP1(CLK := Axis12_BackHome_trigger);
IF UP1.Q THEN M1 := TRUE; Axis12_Negative_Invalid := TRUE; END_IF;
(* Network 2 *)
_p1 := M1 AND NOT Total_Pause;
IF _p1 THEN Axis12_PTF := TRUE; M2 := TRUE; M1 := FALSE; END_IF;
(* Network 3 *)
_p2 := M2 AND Axis12_Negative_Limit;
IF _p2 THEN Axis12_Halt := TRUE; M20 := TRUE; M2 := FALSE; Axis12_PTF := FALSE; END_IF;
(* Network 4 *)
T1(IN := M20 AND Axis12_Halt_Function.Done, PT := T#1MS);
IF T1.Q THEN Axis12_Halt := FALSE; M3 := TRUE; M20 := FALSE; END_IF;
(* Network 5 *)
IF M3 AND NOT Total_Pause THEN M4 := TRUE; Axis12_Home := TRUE; END_IF;
(* Network 6 *)
DOWN1(CLK := M4 AND Axis12_Negative_Limit);
IF DOWN1.Q THEN Axis12_Negative_Invalid := FALSE; END_IF;
(* Network 7 *)
_p3 := M4 AND Axis12_Home_Function.Done;
IF _p3 THEN Axis12_BackHome_OK := TRUE; Axis12_Home := FALSE; Axis12_BackHome_trigger := FALSE; M4 := FALSE; M3 := FALSE; END_IF;
(* Network 8 *)
IF Total_Pause AND Axis12_BackHome_trigger THEN Axis12_Home := FALSE; Axis12_PTF := FALSE; M4 := FALSE; M3 := FALSE; M2 := FALSE; Axis12_Negative_Invalid := TRUE; Axis12_BackHome_OK := FALSE; M1 := TRUE; M20 := FALSE; END_IF;
(* Network 9 *)
(* Network 10 *)
IF Total_Emergency THEN M1 := FALSE; M20 := FALSE; M2 := FALSE; M3 := FALSE; M4 := FALSE; Axis12_BackHome_trigger := FALSE; Axis12_Negative_Invalid := FALSE; Axis12_PTF := FALSE; Axis12_BackHome_OK := FALSE; Axis12_Home := FALSE; END_IF;
(* Network 11 *)
END_PROGRAM

(* POU Other_Folder/Akam_Stop_Message/Initialization_Folder/IniRun, ST *)
PROGRAM IniRun
VAR
	step: INT;
	bak_step:INT;
	rt_hold: R_TRIG;
	M1: BOOL;

	T1: TON;
	T2:TON;


END_VAR

VAR_INPUT
	bstart1: BOOL;
	bhold1: BOOL;
	breset1: BOOL;

END_VAR
(*数据保存*)
IF Save_Button THEN
Save_Par(NETID:='',port:=801,start:=TRUE,tmout:=T#1s);
END_IF
IF NOT Save_Par.BUSY  THEN
Save_Button:=FALSE;
Save_Par(NETID:='',port:=801,start:=FALSE,tmout:=T#1s);
END_IF


(*当出现回原点没有时，需要初始化*)
IF NOT Axis1_BackHome_OK OR NOT  Axis2_BackHome_OK OR NOT Axis3_BackHome_OK OR NOT Axis4_BackHome_OK OR NOT Axis5_BackHome_OK
	OR NOT Axis6_BackHome_OK OR NOT Axis7_BackHome_OK OR NOT Axis8_BackHome_OK OR NOT Axis9_BackHome_OK OR NOT Axis10_BackHome_OK OR NOT Axis11_BackHome_OK  THEN
;(*判断是否需要回原点----------------------------------------------------*)
END_IF
(*---------------------------------------------------------------------------初始化开始流程---------------------------------------------------------------------------------*)
CASE step OF
0:
Need_Ini:=TRUE;(*此时寻妖初始化*)
(*进入初始化流程*)
step:=10;

10:(*判断是否需要初始化*)
IF Need_Ini AND NOT Total_Axis_Error AND NOT Debug_Model   THEN (*当需要初始化的时候，复位所有原点ok信号*)
	Axis1_BackHome_OK:=FALSE;
Axis2_BackHome_OK:=FALSE;
Axis3_BackHome_OK:=FALSE;
Axis4_BackHome_OK:=FALSE;
Axis5_BackHome_OK:=FALSE;
Axis6_BackHome_OK:=FALSE;
Axis7_BackHome_OK:=FALSE;
Axis8_BackHome_OK:=FALSE;
Axis9_BackHome_OK:=FALSE;
Axis10_BackHome_OK:=FALSE;
Axis11_BackHome_OK:=FALSE;
step:=20;
END_IF

20:(*等待复位按钮操作，复位报警等状态*)
IF X4_6 AND Need_Ini THEN
	IF Total_Axis_Error THEN
	M1:=TRUE;(*no use*)(*上位机提示电机报警问题，需要初始化*)
	END_IF
	IF NOT Total_Axis_Error THEN
	step:=30;
	END_IF
END_IF;

30:(*启动按下的处理开始进入初始化过中。。。。。。*)
IF X4_4 AND NOT Total_Axis_Error AND NOT Debug_Model THEN
Need_Ini:=FALSE;
IsIniing:=TRUE;(*初始化中ing*)
M101:=TRUE;(*初始化中，速度为中速*)
Axis1_Poweron:=TRUE;
Axis2_Poweron:=TRUE;
Axis3_Poweron:=TRUE;
Axis4_Poweron:=TRUE;
Axis5_Poweron:=TRUE;
Axis6_Poweron:=TRUE;
Axis7_Poweron:=TRUE;
Axis8_Poweron:=TRUE;
Axis9_Poweron:=TRUE;
Axis10_Poweron:=TRUE;
Axis11_Poweron:=TRUE;
step:=39;
END_IF

39:
(*滑台气缸上下，如果在同一高度，则说明不存在重叠部分，可复位气缸*)
IF (X4_11 AND X4_13) OR (X4_12 AND X4_14)  AND X2_6 THEN
Y1_6:=FALSE;
Y1_7:=FALSE;
step:=40;
ELSE
step:=40;
END_IF


40:(*气缸复位状态保留*)

Y0_2:=FALSE;
Y0_5:=FALSE;
Y0_14:=FALSE;
y0_1:=TRUE;
Y0_12:=FALSE;



(******************** AND  *****************************)

Y0_7:=FALSE;(*左上下气缸*)
Y0_9:=FALSE;(*滚压气缸复位*)
Y1_1:=FALSE;(*右上下气缸*)
Y0_4:=FALSE;
Y1_3:=FALSE;
IF X2_13 AND X3_3 AND X3_11 THEN
	step:=50;(*初步气缸复位*)
END_IF

50:
Y0_6:=FALSE;(*左平移气缸复位*)
Y0_11:=FALSE;(*滚压部分下压气缸复位*)
Y0_16:=FALSE;(*右平移气缸复位*)
T1(IN:=TRUE , PT:=t#1s , Q=> , ET=> );
IF T1.Q AND X2_11 AND X3_9 THEN
T1(IN:=FALSE , PT:=t#1s , Q=> , ET=> );
step:=60;(*无感气缸*)
END_IF

60:(*复位滚压气缸部分气缸，推入气缸，和翻转气缸*)
Y0_10:=FALSE;
IF X3_1 THEN
step:=70;
END_IF

70:(*翻转气缸复位*)
Y0_13:=FALSE;
IF X3_5 THEN
step:=80;
END_IF

80:(*上电延时*)
T2(IN:=TRUE , PT:=t#1s , Q=> , ET=> );
IF T2.Q  AND NOT Total_Pause THEN
T2(IN:=FALSE , PT:=t#1s , Q=> , ET=> );
step:=90;
END_IF

90:
home_backing:=TRUE;
IF NOT Axis3_BackHome_OK OR NOT Axis6_BackHome_OK OR NOT Axis7_BackHome_OK OR NOT Axis8_BackHome_OK OR NOT Axis9_BackHome_OK THEN
step:=100;
ELSE
step:=110;(*当喂料都已经回过原点，则不需要回原点*)
END_IF


100:(*判断是否都需要回原点*)(*喂料部分回原点*)
Axis3_BackHome_trigger:=TRUE;(**)
Axis6_BackHome_trigger:=TRUE;(**)
Axis7_BackHome_trigger:=TRUE;(**)
Axis8_BackHome_trigger:=TRUE;(**)
Axis9_BackHome_trigger:=TRUE;
IF Axis3_BackHome_OK AND Axis6_BackHome_OK AND Axis7_BackHome_OK AND Axis8_BackHome_OK AND Axis9_BackHome_OK  THEN
Axis3_BackHome_trigger:=FALSE;(**)
Axis6_BackHome_trigger:=FALSE;(**)
Axis7_BackHome_trigger:=FALSE;(**)
Axis8_BackHome_trigger:=FALSE;(**)
Axis9_BackHome_trigger:=FALSE;
step:=101;
END_IF

101:(*升降回到初始位置*)
D3:=D300;(*进料初始位置，在下面*)
D6:=D600;(*上升初始位置，在下面*)
D7:=D700;(*下降初始位置，在下面*)
D8:=D800;(*上升初始位置，在下面*)
D9:=D900;(*下降初始位置，在下面*)
Axis3_MoveAbsolute:=TRUE;
Axis6_MoveAbsolute:=TRUE;
Axis7_MoveAbsolute:=TRUE;
Axis8_MoveAbsolute:=TRUE;
Axis9_MoveAbsolute:=TRUE;
IF Axis3_Abs_Function.Done AND Axis6_Abs_Function.Done AND Axis7_Abs_Function.Done AND Axis8_Abs_Function.Done AND Axis9_Abs_Function.Done  THEN
Axis3_MoveAbsolute:=FALSE;
Axis6_MoveAbsolute:=FALSE;
Axis7_MoveAbsolute:=FALSE;
Axis8_MoveAbsolute:=FALSE;
Axis9_MoveAbsolute:=FALSE;
step:=102;  (*初始都在下面*)
END_IF

102:(*Z轴撕膜电机回原*)
Axis5_BackHome_trigger:=TRUE;
IF Axis5_BackHome_OK THEN
Axis5_BackHome_trigger:=FALSE;
step:=103;
END_IF

103:
D5:=A5_W0;(*Z轴回到初始位置*)
Axis5_MoveAbsolute:=TRUE;
IF Axis5_Abs_Function.Done THEN
Axis5_MoveAbsolute:=FALSE;
step:=110;
END_IF

110:(*其余轴回原点*)
Axis1_BackHome_trigger:=TRUE;
Axis11_BackHome_trigger:=TRUE;
Axis2_BackHome_trigger:=TRUE;
Axis4_BackHome_trigger:=TRUE;
Axis10_BackHome_trigger:=TRUE;
IF Axis1_BackHome_OK AND Axis2_BackHome_OK AND Axis4_BackHome_OK  AND Axis10_BackHome_OK AND Axis11_BackHome_OK  THEN
Axis1_BackHome_trigger:=FALSE;
Axis2_BackHome_trigger:=FALSE;
Axis4_BackHome_trigger:=FALSE;
Axis10_BackHome_trigger:=FALSE;
Axis11_BackHome_trigger:=FALSE;
step:=120;
END_IF

120:(*移载等轴的回到初始位置*)
D1:=A1_W0;
D1_1:=A11_W0+250;(*为了保证回原点之后，滑台1气缸在下面，滑台2气缸在上面，则需要，错开初始位置*)
D2:=A2_W0;
D4:=A4_W0;
D10:=A10_W0;
Axis1_MoveAbsolute:=TRUE;
Axis2_MoveAbsolute:=TRUE;
Axis4_MoveAbsolute:=TRUE;
Axis10_MoveAbsolute:=TRUE;
Axis11_MoveAbsolute:=TRUE;
IF Axis1_Abs_Function.Done AND Axis2_Abs_Function.Done AND Axis4_Abs_Function.Done  AND Axis10_Abs_Function.Done AND Axis11_Abs_Function.Done  THEN
Axis1_MoveAbsolute:=FALSE;
Axis2_MoveAbsolute:=FALSE;
Axis4_MoveAbsolute:=FALSE;
Axis10_MoveAbsolute:=FALSE;
Axis11_MoveAbsolute:=FALSE;
home_backing:=FALSE;
Y1_6:=FALSE;(*最终保证，滑台1在上面，滑台2气缸在下面*)
Y1_7:=FALSE;
step:=121;
END_IF


121:
IF  X4_11 AND X4_14 THEN(*最终结果，传感器检测*)
step:=122;
END_IF

122:
D1_1:=A11_W0;
Axis11_MoveAbsolute:=TRUE;
IF  Axis11_Abs_Function.Done THEN
Axis11_MoveAbsolute:=FALSE;
step:=130;
END_IF


130:(*其余需要初始化的状态*)

IsIniing:=FALSE;
Model_Choose:=TRUE;(*模式选择*)
step:=140;

140:
(*模式选选择，直接按钮，启动程序，当选上位机选择调试模式，同时按下启动按钮，则进入调试模式*)
IF NOT Debug_Model AND X4_4 THEN
	Model_Choose:=FALSE;(*模式选择*)
Product_Film_Handel_Run:=TRUE;
Left_Translation_Run_1:=TRUE;
Left_Translation_Run_2:=TRUE;
Right_Translation_Run:=TRUE;
Rolling_Part_Run:=TRUE;
Right_Carry_Run:=TRUE;
Left_Carry_Run:=TRUE;
Liftin_Feed_1_Run:=TRUE;
Liftin_Feed_Left_1_Run:=TRUE;
Liftin_Feed_Left_2_Run:=TRUE;
Liftin_Feed_Right_1_Run:=TRUE;
Liftin_Feed_Right_2_Run:=TRUE;
M102:=TRUE;
Debug_Model:=FALSE;
Positive2_Safe:=TRUE;
	Positive3_Safe:=TRUE;
	Positive_Wait_Safe:=TRUE;
runing:=TRUE;
	step:=150;
END_IF
IF Debug_Model AND X4_4 THEN
	M100:=TRUE;(*调试模式下低速*)
	Model_Choose:=FALSE;(*模式选择*)
	Axis1_debug_trigger:=TRUE;
Axis1_debug_trigger:=TRUE;
Axis2_debug_trigger:=TRUE;
Axis3_debug_trigger:=TRUE;
Axis4_debug_trigger:=TRUE;
Axis5_debug_trigger:=TRUE;
Axis6_debug_trigger:=TRUE;
Axis7_debug_trigger:=TRUE;
Axis8_debug_trigger:=TRUE;
Axis9_debug_trigger:=TRUE;
Axis10_debug_trigger:=TRUE;
Axis11_debug_trigger:=TRUE;
(*其余调试模式*)
 step:=160;
END_IF

150:(*运行模式下的死循环*)
;


160:
(*调试模式下的死循环，等待调试模式借宿，重新开始初始化*)
IF NOT Debug_Model THEN
Need_Ini:=TRUE;
 	    bak_step:=0;
	step:=0;
END_IF



300:(*外部输入启动*)
    IF bstart1   AND NOT Total_Axis_Error AND NOT total_pausestatus THEN
	step:=bak_step;
END_IF;
END_CASE;



(*触发暂停的外部输入*)
rt_hold(CLK:=( Total_Axis_Error OR  bhold1) , Q=> ); (*暂停状态*)
IF step<>0 AND step<>300   AND  rt_hold.Q THEN
     bak_step:=step;
     step:=300;
END_IF

(*急停处理*)
IF Total_Emergency THEN
debug_FLIG:=FALSE;
M100:=FALSE;
M101:=FALSE;
M102:=FALSE;
IsIniing:=FALSE;
runing:=FALSE;
home_backing:=FALSE;
Model_Choose:=FALSE;(*模式选择*)


Debug_Model:=FALSE;
Positive2_Safe:=FALSE;
Positive3_Safe:=FALSE;
Positive_Wait_Safe:=FALSE;


bak_step:=0;
step:=0;
END_IF


(*与debug1中的梯形图一起使用，当不在应该调试模式下的时候，按下调试按钮，自动复位--------详见------debug1----------*)
IF step<>160 AND step<>140 AND step<>300  THEN
debug_FLIG:=FALSE;
ELSE
debug_FLIG:=TRUE;
END_IF
END_PROGRAM

(* POU old/Old_Tray_Pro/Liftin_Feed_Right_1, ST *)
PROGRAM Liftin_Feed_Right_1
VAR

	step: INT;
	bak_step:INT;
	rt_hold: R_TRIG;
	UP1: R_TRIG;
	T1: TON;
	T2:TON;

END_VAR

VAR_INPUT
	bstart1: BOOL;
	bhold1: BOOL;
	breset1: BOOL;

END_VAR
UP1(CLK:=Liftin_Feed_Right_1_Run , Q=> );

CASE step OF
0:
 IF UP1.Q THEN
step:=10;
END_IF


10:(*上升运行*)
Axis8_PTF_2:=TRUE;
IF X2_4 AND  X1_3 THEN(*碰到光纤，同时没有碰到极限，此时上料ok*)
Axis8_PTF_2:=FALSE;
Feed_3_Finish:=TRUE;
Axis8_Halt:=TRUE;
step:=20;
END_IF
IF NOT X1_3 THEN(*碰到极限，此时表示料空*)
Axis8_PTF_2:=FALSE;
Axis8_Halt:=TRUE;
step:=50;
END_IF

20:
Axis8_Halt:=FALSE;
(*表示上料成功,等待取完信号*)
IF Get_Robort3_Tray_Full THEN
Feed_3_Finish:=FALSE;
Get_Robort3_Tray_Full:=FALSE;(*放满信号，给出，等待移动*)
Right_Can_Move:=TRUE;
step:=30;
END_IF


30:(*等待平移完成，才可以上升*)
IF Right_Move_Finish THEN
Right_Move_Finish:=FALSE;
step:=10;
END_IF


50:(*碰到极限，此时料取完,回到初始位置*)
Axis8_Halt:=FALSE;
D8:=D800;
Axis8_MoveAbsolute:=TRUE;
IF Axis8_Abs_Function.Done THEN
Axis8_MoveAbsolute:=FALSE;
Feed_Right_None_Alam:=TRUE;(*不暂停，只提示*)
step:=60;
END_IF

60:(*回到初始位置，提示料空*)
IF Right_UP_Button AND NOT Total_Pause THEN
Right_UP_Button:=FALSE;
Feed_Right_None_Alam:=FALSE;(*不暂停，只提示*)
step:=10;
END_IF

300:
    IF bstart1   AND NOT Total_Axis_Error AND NOT total_pausestatus THEN
	step:=bak_step;
END_IF;
END_CASE


rt_hold(CLK:=( Total_Axis_Error OR  bhold1) , Q=> ); (*暂停状态*)
IF step<>0 AND step<>300   AND  rt_hold.Q THEN
     bak_step:=step;
     step:=300;
END_IF


IF Right_UP_Button THEN
Right_UP_Button:=FALSE;
END_IF

IF Total_Emergency THEN
Liftin_Feed_Right_1_Run:=FALSE;
Feed_Right_None_Alam:=FALSE;
Feed_3_Finish:=FALSE;


bak_step:=0;
step:=0;
END_IF


(*随时可以不做料的操作*)
IF Feed_Right_Button1 AND step=20 AND NOT Total_Pause THEN
Feed_Right_Button1:=FALSE;
Feed_3_Finish:=FALSE;
step:=50;
ELSE
Feed_Right_Button1:=FALSE;
END_IF
END_PROGRAM

(* POU old/Old_Tray_Pro/Liftin_Feed_Right_2, ST *)
PROGRAM Liftin_Feed_Right_2
VAR

	step: INT;
	bak_step:INT;
	rt_hold: R_TRIG;
	UP1: R_TRIG;
	DOWN1: F_TRIG;

	T1: TON;
	T2:TON;

END_VAR

VAR_INPUT
	bstart1: BOOL;
	bhold1: BOOL;
	breset1: BOOL;

END_VAR
(*左下降，初始化，回原点到初始位置，，，启动之后，先往上走，到初始位置(第一次回原点使用)  ，接收到送料完成可下降信号，则
开始下降，等现将结束，告知，可放料*)

UP1(CLK:=Liftin_Feed_Right_2_Run , Q=> );

CASE step OF
0:
 IF UP1.Q THEN
step:=1;
END_IF

1:
(*初始化之后位置在下面的初始位置*)
Axis9_PTF_2:=TRUE;
IF X2_5 AND X1_6 THEN
Axis9_PTF_2:=FALSE;
Axis9_Halt:=TRUE;
step:=20;
END_IF
IF NOT X1_6 THEN
Axis9_PTF_2:=FALSE;
Axis9_Halt:=TRUE;
step:=60;(*撞到极限，此时需要回到上面的初始位置*)
END_IF

10:
(*初始化的时候写，回原点之后，向上跑知道碰到光纤，或者极限的时候，到极限回到初始位置，碰到光纤，停止，翻转到极限停止位置*)

(*到初始位置，等待放料，当光纤感应到，同时，接收到，可下降信号的时候，开始下降，当感应不到光纤，则停止*)
IF you_ke_jiang AND X2_5 THEN
you_ke_jiang:=FALSE;
	step:=20;
END_IF

20:
Axis9_Halt:=FALSE;
(*接收到可降信号，开始下降，到传感器下降沿停止下降，等待*)
Axis9_PTF:=TRUE;
DOWN1(CLK:=X2_5 , Q=> );
IF DOWN1.Q AND NOT  X1_7 THEN
Axis9_PTF:=FALSE;
you_down_Finish:=TRUE;
Axis9_Halt:=TRUE;
step:=30;
END_IF
IF  X1_7 THEN(*碰到极限，此时表示料空*)
Axis9_PTF:=FALSE;
Axis9_Halt:=TRUE;
step:=400;
END_IF

30:(*停止，给出下降完成信号，等待放料循环*)
Axis9_Halt:=FALSE;
step:=10;

400:(*碰到原点，此时，回到下初始位置，给出料满提示*)
Axis9_Halt:=FALSE;
D9:=D900;
Axis9_MoveAbsolute:=TRUE;
IF Axis9_Abs_Function.Done THEN
Axis9_MoveAbsolute:=FALSE;
Feed_Right_None_Alam:=TRUE;(*不暂停，只提示*)
step:=50;
END_IF

50:(*碰到下极限，给出缺料提示*)
Axis9_Halt:=FALSE;
IF Right_Down_Button AND NOT Total_Pause THEN
	Right_Down_Button:=FALSE;
Feed_Right_Full_Alam:=FALSE;
	step:=1;(*确认拿走料之后，运动到初始位置*)
END_IF

60:(*回到初始位置*)
Axis9_Halt:=FALSE;
D9:=D910;
Axis9_MoveAbsolute:=TRUE;
IF Axis9_Abs_Function.Done THEN
Axis9_MoveAbsolute:=FALSE;
you_down_Finish:=TRUE;(*左下降完成信号*)
step:=10;
END_IF

300:
    IF bstart1   AND NOT Total_Axis_Error AND NOT total_pausestatus THEN
	step:=bak_step;
END_IF;
END_CASE


rt_hold(CLK:=( Total_Axis_Error OR  bhold1) , Q=> ); (*暂停状态*)
IF step<>0 AND step<>300   AND  rt_hold.Q THEN
     bak_step:=step;
     step:=300;
END_IF


IF Total_Emergency THEN
Liftin_Feed_Right_2_Run:=FALSE;
you_down_Finish:=FALSE;
Feed_Right_Full_Alam:=FALSE;


bak_step:=0;
step:=0;
END_IF


(*随时可以不做料的操作*)
IF Feed_Right_Button2 AND step=10 AND NOT Total_Pause THEN
Feed_Right_Button2:=FALSE;
you_down_Finish:=FALSE;
step:=400;
ELSE
Feed_Right_Button2:=FALSE;
END_IF
END_PROGRAM

(* POU Test_Part_pro/New_Table_3, ST *)
PROGRAM New_Table_3
VAR
	step: INT;
	bak_step:INT;
	rt_hold: R_TRIG;
	UP1: R_TRIG;
	Run_Time:BOOL;
	T1:TON;
	Run_Time_Lreal: TIME;




	T2: TON;
	T3: TON;
END_VAR

VAR_INPUT
	bstart1: BOOL;
	bhold1: BOOL;
	breset1: BOOL;

END_VAR
UP1(CLK:=Left_Translation_Run_2 , Q=> );

CASE step OF
0:
 IF UP1.Q THEN
step:=10;
END_IF

10:
D1_1:=A11_W1;(*左等待放料工位*)
Axis11_MoveAbsolute:=TRUE;
IF Axis11_Abs_Function.Done THEN
Axis11_MoveAbsolute:=FALSE;
step:=20;
END_IF;

20:(*到下初始位置------寻味位置1是否安全*)
IF Positive1_Safe THEN
	Positive1_Safe:=FALSE;
	Y1_7:=TRUE;
step:=30;
END_IF

30:
IF X4_13 THEN
	Positive4_Safe:=TRUE;
	step:=40;
END_IF

40:(*安全之后上顶*)
IF Tray2_Have THEN
	step:=72;
ELSE
step:=72;
END_IF

50:(*到位置之后，告知可以放料*)
D1_1:=A11_W1;(*左等待放料工位*)
Axis11_MoveAbsolute:=TRUE;
IF Axis11_Abs_Function.Done THEN
Process_2_Can_Push:=TRUE;
Axis11_MoveAbsolute:=FALSE;
Y0_2:=TRUE;
step:=60;
END_IF;

60:(*上料-----等待放下之后---------*)
IF Process_1_Push_Finish THEN
Tray2_Have:=TRUE;
Process_1_Push_Finish:=FALSE;
step:=70;
END_IF

70:
T2(IN:=TRUE , PT:=t#1s , Q=> , ET=> );
   IF T2.Q AND NOT Total_Pause  THEN
T2(IN:=FALSE, PT:=t#1S , Q=> , ET=> );
Can_Move_Film:=TRUE;(*给出可撕膜信号*)
step:=71;
END_IF

71:(*撕膜完成信号等到*)
IF Process_1_Push_Finish_Sure THEN
Process_1_Push_Finish_Sure:=FALSE;
step:=72;
END_IF

72:(*判断拍照位置1是否安全*)
IF Positive_Camera_Safe1 THEN
Positive_Camera_Safe1:=FALSE;(*拍照位置1被占据*)
step:=73;
END_IF

73:
D1_1:=A11_W2;(*拍照工位1*)
Axis11_MoveAbsolute:=TRUE;
IF Axis11_Abs_Function.Done THEN
Axis11_MoveAbsolute:=FALSE;
(*到位拍照*)
step:=90;
END_IF

80:(*拍照工位1拍照结束-----等待*)
IF Camera_1_5_OK THEN
Camera_1_5_run:=FALSE;
Camera_1_5_OK:=FALSE;
step:=90;
END_IF
IF Camera1_NG THEN  (*拍照失败的处理，判断ng,此时需要给出结果，，，，，，，同时运动到工作位置*)
Camera_1_5_run:=FALSE;
Tray2_Have:=FALSE;
Camera1_NG:=FALSE;
Y0_2:=FALSE;
step:=2000;
END_IF

90:(*判断拍照位置2是否安全*)
IF Positive_Camera_Safe2 THEN
Positive_Camera_Safe2:=FALSE;
step:=100;
END_IF

100:(*移动到位置2*)
D1_1:=A11_W3; (*拍照工位2*)
Axis11_MoveAbsolute:=TRUE;
IF Axis11_Abs_Function.Done THEN
Axis11_MoveAbsolute:=FALSE;
(*到位拍照*)
step:=120;
END_IF

110:
IF Camera_1_6_OK THEN
Camera_1_6_run:=FALSE;
Camera_1_6_OK:=FALSE;
step:=120;
END_IF
IF Camera1_NG THEN  (*拍照失败的处理，判断ng,此时需要给出结果，，，，，，，同时运动到工作位置*)
Camera_1_6_run:=FALSE;
Tray2_Have:=FALSE;
Camera1_NG:=FALSE;
Y0_2:=FALSE;
step:=2020;
END_IF


120:(*判断位置3是否安全*)
IF Positive_Camera_Safe3 THEN
Positive_Camera_Safe3:=FALSE;
step:=130;
END_IF

130:(*到工位3*)
D1_1:=A11_W4;(*拍照工位3*)
Axis11_MoveAbsolute:=TRUE;
IF Axis11_Abs_Function.Done THEN
Axis11_MoveAbsolute:=FALSE;
(*到位拍照*)
step:=150;
END_IF

140:
IF Camera_1_7_OK THEN
Camera_1_7_run:=FALSE;
Camera_1_7_OK:=FALSE;
step:=150;
END_IF
IF Camera1_NG THEN  (*拍照失败的处理，判断ng,此时需要给出结果，，，，，，，同时运动到工作位置*)
Camera_1_7_run:=FALSE;
Tray2_Have:=FALSE;
Camera1_NG:=FALSE;
Y0_2:=FALSE;
step:=2050;
END_IF

150:(*拍照位置3判断是否安全----------*)
IF Positive_Camera_Safe4 THEN
Positive_Camera_Safe4:=FALSE;
step:=160;
END_IF

160:
D1_1:=A11_W5;(*拍照工位4*)
Axis11_MoveAbsolute:=TRUE;
IF Axis11_Abs_Function.Done THEN
Axis11_MoveAbsolute:=FALSE;
(*到位拍照*)

Positive1_Safe:=TRUE;
step:=180;
END_IF

170:
IF Camera_1_8_OK THEN
Camera_1_8_run:=FALSE;
Camera_1_8_OK:=FALSE;
step:=180;
END_IF
IF Camera1_NG THEN  (*拍照失败的处理，判断ng,此时需要给出结果，，，，，，，同时运动到工作位置*)
Camera_1_8_run:=FALSE;
Tray2_Have:=FALSE;
Camera1_NG:=FALSE;
Y0_2:=FALSE;
step:=2070;
END_IF

180:(*判断工作位置1是否安全*)
IF Positive_Fit_Safe1 THEN
Positive_Fit_Safe1:=FALSE;
(*
HB_Fit_Finish_5:=FALSE;
HB_Fit_Finish_6:=FALSE;
HB_Fit_Finish_7:=FALSE;
HB_Fit_Finish_8:=FALSE;*)
step:=190;
END_IF

190:(*到工作位置1*)
D1_1:=A11_W6;(*工作位置工位1*)
Axis11_MoveAbsolute:=TRUE;
IF Axis11_Abs_Function.Done THEN
Axis11_MoveAbsolute:=FALSE;

Positive_Camera_Safe1:=TRUE;(*工作位置1是给出拍照位置1安全安全位置-------------------------------------*)

step:=210;
END_IF

200:(*到位等待贴合完成*)
IF HB_Fit_Finish_5 THEN
FG_Ready_5:=FALSE;
HB_Fit_Finish_5:=FALSE;
step:=210;
END_IF

210:(*工位1贴合完成-----询问工作位置2是否安全*)
IF Positive_Fit_Safe2 THEN
Positive_Fit_Safe2:=FALSE;
step:=220;
END_IF

220:(*位置安全------到贴合位置2*)
D1_1:=A11_W7;(*工作位置工位1*)
Axis11_MoveAbsolute:=TRUE;
IF Axis11_Abs_Function.Done THEN
Axis11_MoveAbsolute:=FALSE;

Positive_Camera_Safe2:=TRUE;(*工作位置1是给出拍照位置1安全安全位置-------------------------------------*)

step:=240;
END_IF

230:(*等待贴合完成信号*)
IF HB_Fit_Finish_6 THEN
FG_Ready_6:=FALSE;
HB_Fit_Finish_6:=FALSE;
step:=240;
END_IF

240:(*贴合完成------寻问位置3是否安全*)
IF Positive_Fit_Safe3 THEN
Positive_Fit_Safe3:=FALSE;
step:=250;
END_IF

250:(*位置安全------到贴合位置2*)
D1_1:=A11_W8;(*工作位置工位1*)
Axis11_MoveAbsolute:=TRUE;
IF Axis11_Abs_Function.Done THEN
Axis11_MoveAbsolute:=FALSE;

Positive_Camera_Safe3:=TRUE;(*工作位置1是给出拍照位置1安全安全位置-------------------------------------*)

step:=270;
END_IF

260:(*等待贴合完成信号*)
IF HB_Fit_Finish_7 THEN
FG_Ready_7:=FALSE;
HB_Fit_Finish_7:=FALSE;
step:=270;
END_IF

270:(*位置3贴合完成，询问位置4是否安全*)
IF Positive_Fit_Safe4 THEN
Positive_Fit_Safe4:=FALSE;
step:=280;
END_IF

280:(*位置安全------到贴合位置2*)
D1_1:=A11_W9;(*工作位置工位1*)
Axis11_MoveAbsolute:=TRUE;
IF Axis11_Abs_Function.Done THEN
Axis11_MoveAbsolute:=FALSE;

Positive_Camera_Safe4:=TRUE;(*工作位置1是给出拍照位置1安全安全位置-------------------------------------*)

step:=300;
END_IF

